(* CODESYS project P_ruwdkj.project
   Title: B_Ugol
   Version: 0.0.0.0

Project tree, tasks and I/O mapping:
  MyController : TM241CEC24T/U, Schneider Electric, order no. TM241CEC24T/U, version 4.0.5.9
    application Application
      task MAST (cyclic, interval 20 ms, priority 15, watchdog 100 ms x 1) calls POU_Hand, POU_Auto, POU_Out, POU_Alarm, POU_testing
      global variables GVL
      program POU_Hand [LD]
      program POU_Out [LD]
      program POU_Auto [LD]
      Symbols
      program POU_Alarm [LD]
      program POU_testing [LD]
    DI : Digital Inputs, Schneider Electric, version 4.0.5.9
        input  iwDI_IW0 : WORD  // IW0
        input  i_AvStop : BOOL  // IW0.I0
        input  i_TZ_K1 : BOOL  // IW0.I1
        input  i_TZ_KR2 : BOOL  // IW0.I2
        input  i_Tros_K1 : BOOL  // IW0.I3
        input  i_Tros_KR2 : BOOL  // IW0.I4
        input  i_Di_Rezerv1 : BOOL  // IW0.I5
        input  i_Di_Rezerv2 : BOOL  // IW0.I6
        input  i_Di_Rezerv3 : BOOL  // IW0.I7
        input  i_Di_Rezerv4 : BOOL  // IW0.I8
        input  i_Di_Rezerv5 : BOOL  // IW0.I9
        input  i_Di_Rezerv6 : BOOL  // IW0.I10
        input  i_Di_Rezerv7 : BOOL  // IW0.I11
        input  i_Di_Rezerv8 : BOOL  // IW0.I12
        input  i_Di_Rezerv9 : BOOL  // IW0.I13
        input  ibDI_IB1 : BYTE  // IB1
    DQ : Digital Outputs, Schneider Electric, version 4.0.5.9
        output q_PuskK1 : BOOL  // QW0.Q0
        output q_PuskEP80 : BOOL  // QW0.Q1
        output q_PuskKR2_for : BOOL  // QW0.Q2
        output q_PuskKR2_rev : BOOL  // QW0.Q3
        output q_Zvonok : BOOL  // QW0.Q4
        output q_Red1 : BOOL  // QW0.Q5
        output q_Yellow1 : BOOL  // QW0.Q6
        output q_Green1 : BOOL  // QW0.Q7
        output q_Red2 : BOOL  // QW0.Q8
        output q_Yellow2 : BOOL  // QW0.Q9
        output qbDQ_QB1 : BYTE  // QB1
        unmapped channels: QW0
    Counters : Counters, Schneider Electric, version 4.0.5.9
    Pulse_Generators : Pulse Generators, Schneider Electric, version 4.0.5.9
    Cartridge_1 : Cartridge, Schneider Electric, version 4.0.5.9
    IO_Bus : IO bus - TM3, Schneider Electric, version 4.0.5.9
      Module_1 : TM3DQ8T/G, Schneider Electric, order no. TM3DQ8T/G, version 1.0.1.3
          output q_Green2 : BOOL  // QB0.Q0
          output q_Dq_Rezerv1 : BOOL  // QB0.Q1
          output q_Dq_Rezerv2 : BOOL  // QB0.Q2
          output q_Dq_Rezerv3 : BOOL  // QB0.Q3
          output q_Dq_Rezerv4 : BOOL  // QB0.Q4
          output q_Dq_Rezerv5 : BOOL  // QB0.Q5
          output q_Dq_Rezerv6 : BOOL  // QB0.Q6
          output q_Dq_Rezerv7 : BOOL  // QB0.Q7
          unmapped channels: QB0
      Module_2 : TM3AI8/G, Schneider Electric, order no. TM3AI8/G, version 1.0.0.16
          settings: KPI Configuration.KPI Configuration[0] = 35; KPI Configuration.KPI Configuration[1] = 35; KPI Configuration.KPI Configuration[2] = 35; KPI Configuration.KPI Configuration[3] = 35; KPI Configuration.KPI Configuration[8] = 160; KPI Configuration.KPI Configuration[9] = 15; KPI Configuration.KPI Configuration[10] = 160; KPI Configuration.KPI Configuration[11] = 15; KPI Configuration.KPI Configuration[12] = 160; KPI Configuration.KPI Configuration[13] = 15; KPI Configuration.KPI Configuration[14] = 160; KPI Configuration.KPI Configuration[15] = 15; KPI Configuration.KPI Configuration[24] = 32; KPI Configuration.KPI Configuration[25] = 78; KPI Configuration.KPI Configuration[26] = 32; KPI Configuration.KPI Configuration[27] = 78; KPI Configuration.KPI Configuration[28] = 32; KPI Configuration.KPI Configuration[29] = 78; KPI Configuration.KPI Configuration[30] = 32; KPI Configuration.KPI Configuration[31] = 78
          input  i_Uroven111 : INT  // IW0
          input  i_Uroven112 : INT  // IW1
          input  i_Uroven3 : INT  // IW2
          input  i_Uroven4 : INT  // IW3
          input  iiModule_2_IW4 : INT  // IW4
          input  iiModule_2_IW5 : INT  // IW5
          input  iiModule_2_IW6 : INT  // IW6
          input  iiModule_2_IW7 : INT  // IW7
          input  ibModule_2_IBStatusIW0 : BYTE  // IBStatusIW0
          input  ibModule_2_IBStatusIW1 : BYTE  // IBStatusIW1
          input  ibModule_2_IBStatusIW2 : BYTE  // IBStatusIW2
          input  ibModule_2_IBStatusIW3 : BYTE  // IBStatusIW3
          input  ibModule_2_IBStatusIW4 : BYTE  // IBStatusIW4
          input  ibModule_2_IBStatusIW5 : BYTE  // IBStatusIW5
          input  ibModule_2_IBStatusIW6 : BYTE  // IBStatusIW6
          input  ibModule_2_IBStatusIW7 : BYTE  // IBStatusIW7
    COM_Bus : COM bus, Schneider Electric, version 4.0.5.9
    Ethernet_1 : Ethernet Network, Schneider Electric, version 4.0.5.9
    Serial_Line_1 : Serial line, Schneider Electric, version 4.0.5.9
      SoMachine_Network_Manager : SoMachine-Network Manager, Schneider Electric, version 4.0.0.2
    Serial_Line_2 : Serial line, Schneider Electric, version 4.0.5.9
      Modbus_Manager : Modbus Manager, Schneider Electric, version 4.0.0.2
    CAN_1 : CANopen bus, Schneider Electric, version 4.0.5.9
      CANopen_Performance : CANopen Performance, Schneider Electric, order no. 1806, version 3.0.1.24
          settings: ConfigVersion = 50659584
        Pitatel1 : Altivar 312, Schneider Electric, order no. 0, version 4.5.0.0
            settings: General Options.Optional Device = TRUE; NODEIDSAVED = 1; SDO Timeout = 1000000; Explicit Deactivate PDOs = FALSE; EXPERTSETTINGS = True; Heartbeat-Producer Time = 200; PDO 16#1405.COBID = 16#0301; PDO 16#1805.COBID = 16#0281; Heartbeat-Consuming1.Heartbeat-Time = 300 ms; Drivecom command reg..Subindex = 16#00; Drivecom command reg..Subindex = 16#00; Frequency Reference.Subindex = 16#03; Target velocity.Index = 16#6042; Target velocity.Subindex = 16#00; Target velocity.ObjectLength = 16; Drivecom status register.Subindex = 16#00; Drivecom status register.Subindex = 16#00; Output frequency.Index = 16#2002; Output frequency.Subindex = 16#03; Output frequency.ObjectLength = 16; Motor Current.Index = 16#2002; Motor Current.Subindex = 16#05; Motor Current.ObjectLength = 16; SDO List.Set Guardtime.Index = 16#100C; SDO List.Set Guardtime.Subindex = 16#00; SDO List.Set Guardtime.Value = 16#00000000; SDO List.Set Guardtime.Size = 16; SDO List.Set Guardtime.AbortIfError = FALSE; SDO List.Set Guardtime.JumpToLine = FALSE; SDO List.Set Guardtime.Line = 0; SDO List.Set Lifetime.Index = 16#100D; SDO List.Set Lifetime.Subindex = 16#00; SDO List.Set Lifetime.Value = 16#00000000; SDO List.Set Lifetime.Size = 8; SDO List.Set Lifetime.AbortIfError = FALSE; SDO List.Set Lifetime.JumpToLine = FALSE; SDO List.Set Lifetime.Line = 0; SDO List.Set Heartbeat Consumer.Index = 16#1016; SDO List.Set Heartbeat Consumer.Subindex = 16#01; SDO List.Set Heartbeat Consumer.Value = 16#007F012C;
              SDO List.Set Heartbeat Consumer.Size = 32; SDO List.Set Heartbeat Consumer.AbortIfError = FALSE; SDO List.Set Heartbeat Consumer.JumpToLine = FALSE; SDO List.Set Heartbeat Consumer.Line = 0; SDO List.Set Heartbeat Producer.Index = 16#1017; SDO List.Set Heartbeat Producer.Subindex = 16#00; SDO List.Set Heartbeat Producer.Value = 16#000000C8; SDO List.Set Heartbeat Producer.Size = 16; SDO List.Set Heartbeat Producer.AbortIfError = FALSE; SDO List.Set Heartbeat Producer.JumpToLine = FALSE; SDO List.Set Heartbeat Producer.Line = 0; SDO List.Disable PDO.Index = 16#1400; SDO List.Disable PDO.Subindex = 16#01; SDO List.Disable PDO.Value = 16#80000201; SDO List.Disable PDO.Size = 32; SDO List.Disable PDO.AbortIfError = FALSE; SDO List.Disable PDO.JumpToLine = FALSE; SDO List.Disable PDO.Line = 0; SDO List.Disable PDO.Index = 16#1405; SDO List.Disable PDO.Subindex = 16#01; SDO List.Disable PDO.Value = 16#80000301; SDO List.Disable PDO.Size = 32; SDO List.Disable PDO.AbortIfError = FALSE; SDO List.Disable PDO.JumpToLine = FALSE; SDO List.Disable PDO.Line = 0; SDO List.Set transmission type.Index = 16#1405; SDO List.Set transmission type.Subindex = 16#02; SDO List.Set transmission type.Value = 16#FF; SDO List.Set transmission type.Size = 8; SDO List.Set transmission type.AbortIfError = FALSE; SDO List.Set transmission type.JumpToLine = FALSE; SDO List.Set transmission type.Line = 0; SDO List.Clear pdo mapping.Index = 16#1605; SDO List.Clear pdo mapping.Subindex = 16#00; SDO List.Clear pdo mapping.Value = 16#0; SDO List.Clear pdo mapping.Size = 8; SDO List.Clear pdo mapping.AbortIfError = FALSE; SDO List.Clear pdo mapping.JumpToLine = FALSE; SDO List.Clear pdo mapping.Line = 0; SDO List.Set Mapping.Index = 16#1605;
              SDO List.Set Mapping.Subindex = 16#01; SDO List.Set Mapping.Value = 16#60400010; SDO List.Set Mapping.Size = 32; SDO List.Set Mapping.AbortIfError = FALSE; SDO List.Set Mapping.JumpToLine = FALSE; SDO List.Set Mapping.Line = 0; SDO List.Set Mapping.Index = 16#1605; SDO List.Set Mapping.Subindex = 16#02; SDO List.Set Mapping.Value = 16#20370310; SDO List.Set Mapping.Size = 32; SDO List.Set Mapping.AbortIfError = FALSE; SDO List.Set Mapping.JumpToLine = FALSE; SDO List.Set Mapping.Line = 0; SDO List.Set Mapping.Index = 16#1605; SDO List.Set Mapping.Subindex = 16#03; SDO List.Set Mapping.Value = 16#60420010; SDO List.Set Mapping.Size = 32; SDO List.Set Mapping.AbortIfError = FALSE; SDO List.Set Mapping.JumpToLine = FALSE; SDO List.Set Mapping.Line = 0; SDO List.Set number of pdos.Index = 16#1605; SDO List.Set number of pdos.Subindex = 16#00; SDO List.Set number of pdos.Value = 16#03; SDO List.Set number of pdos.Size = 8; SDO List.Set number of pdos.AbortIfError = FALSE; SDO List.Set number of pdos.JumpToLine = FALSE; SDO List.Set number of pdos.Line = 0; SDO List.Set and enable COB-ID.Index = 16#1405; SDO List.Set and enable COB-ID.Subindex = 16#01; SDO List.Set and enable COB-ID.Value = 16#00000301; SDO List.Set and enable COB-ID.Size = 32; SDO List.Set and enable COB-ID.AbortIfError = FALSE; SDO List.Set and enable COB-ID.JumpToLine = FALSE; SDO List.Set and enable COB-ID.Line = 0; SDO List.Disable PDO.Index = 16#1800; SDO List.Disable PDO.Subindex = 16#01; SDO List.Disable PDO.Value = 16#80000181; SDO List.Disable PDO.Size = 32; SDO List.Disable PDO.AbortIfError = FALSE; SDO List.Disable PDO.JumpToLine = FALSE;
              SDO List.Disable PDO.Line = 0; SDO List.Disable PDO.Index = 16#1805; SDO List.Disable PDO.Subindex = 16#01; SDO List.Disable PDO.Value = 16#80000281; SDO List.Disable PDO.Size = 32; SDO List.Disable PDO.AbortIfError = FALSE; SDO List.Disable PDO.JumpToLine = FALSE; SDO List.Disable PDO.Line = 0; SDO List.Set transmission type.Index = 16#1805; SDO List.Set transmission type.Subindex = 16#02; SDO List.Set transmission type.Value = 16#FF; SDO List.Set transmission type.Size = 8; SDO List.Set transmission type.AbortIfError = FALSE; SDO List.Set transmission type.JumpToLine = FALSE; SDO List.Set transmission type.Line = 0; SDO List.Set inhibit time.Index = 16#1805; SDO List.Set inhibit time.Subindex = 16#03; SDO List.Set inhibit time.Value = 16#001E; SDO List.Set inhibit time.Size = 16; SDO List.Set inhibit time.AbortIfError = FALSE; SDO List.Set inhibit time.JumpToLine = FALSE; SDO List.Set inhibit time.Line = 0; SDO List.Set event time.Index = 16#1805; SDO List.Set event time.Subindex = 16#05; SDO List.Set event time.Value = 16#0064; SDO List.Set event time.Size = 16; SDO List.Set event time.AbortIfError = FALSE; SDO List.Set event time.JumpToLine = FALSE; SDO List.Set event time.Line = 0; SDO List.Clear pdo mapping.Index = 16#1A05; SDO List.Clear pdo mapping.Subindex = 16#00; SDO List.Clear pdo mapping.Value = 16#0; SDO List.Clear pdo mapping.Size = 8; SDO List.Clear pdo mapping.AbortIfError = FALSE; SDO List.Clear pdo mapping.JumpToLine = FALSE; SDO List.Clear pdo mapping.Line = 0; SDO List.Set Mapping.Index = 16#1A05; SDO List.Set Mapping.Subindex = 16#01; SDO List.Set Mapping.Value = 16#60410010; SDO List.Set Mapping.Size = 32;
              SDO List.Set Mapping.AbortIfError = FALSE; SDO List.Set Mapping.JumpToLine = FALSE; SDO List.Set Mapping.Line = 0; SDO List.Set Mapping.Index = 16#1A05; SDO List.Set Mapping.Subindex = 16#02; SDO List.Set Mapping.Value = 16#20020310; SDO List.Set Mapping.Size = 32; SDO List.Set Mapping.AbortIfError = FALSE; SDO List.Set Mapping.JumpToLine = FALSE; SDO List.Set Mapping.Line = 0; SDO List.Set Mapping.Index = 16#1A05; SDO List.Set Mapping.Subindex = 16#03; SDO List.Set Mapping.Value = 16#20020510; SDO List.Set Mapping.Size = 32; SDO List.Set Mapping.AbortIfError = FALSE; SDO List.Set Mapping.JumpToLine = FALSE; SDO List.Set Mapping.Line = 0; SDO List.Set number of pdos.Index = 16#1A05; SDO List.Set number of pdos.Subindex = 16#00; SDO List.Set number of pdos.Value = 16#03; SDO List.Set number of pdos.Size = 8; SDO List.Set number of pdos.AbortIfError = FALSE; SDO List.Set number of pdos.JumpToLine = FALSE; SDO List.Set number of pdos.Line = 0; SDO List.Set and enable COB-ID.Index = 16#1805; SDO List.Set and enable COB-ID.Subindex = 16#01; SDO List.Set and enable COB-ID.Value = 16#00000281; SDO List.Set and enable COB-ID.Size = 32; SDO List.Set and enable COB-ID.AbortIfError = FALSE; SDO List.Set and enable COB-ID.JumpToLine = FALSE; SDO List.Set and enable COB-ID.Line = 0; ConfigVersion = 50659584
            output q_ATVPit1_Controlword : UINT  // Drivecom command reg.
            output qiAltivar_312_1_Frequency_Reference : INT  // Frequency Reference
            output q_ATVPit1_WriteVelocity : INT  // Target velocity
            input  i_ATVPit1_Status : UINT  // Drivecom status register
            input  i_ATVPit1_OutFrec : INT  // Output frequency
            input  i_ATVPit1_OutCur : UINT  // Motor Current
        Pitatel2 : Altivar 312, Schneider Electric, order no. 0, version 4.5.0.0
            settings: General Options.Optional Device = TRUE; NODEIDSAVED = 3; SDO Timeout = 1000000; Explicit Deactivate PDOs = FALSE; EXPERTSETTINGS = True; Emergency-General Parameters.Emergency COBID = 16#83; Heartbeat-Producer Time = 200; PDO 16#1400.COBID = 16#80000203; PDO 16#1405.COBID = 16#0303; PDO 16#1800.COBID = 16#80000183; PDO 16#1805.COBID = 16#0283; Heartbeat-Consuming1.Heartbeat-Time = 300 ms; Drivecom command reg..Subindex = 16#00; Drivecom command reg..Subindex = 16#00; Frequency Reference.Subindex = 16#03; Target velocity.Index = 16#6042; Target velocity.Subindex = 16#00; Target velocity.ObjectLength = 16; Drivecom status register.Subindex = 16#00; Drivecom status register.Subindex = 16#00; Output frequency.Index = 16#2002; Output frequency.Subindex = 16#03; Output frequency.ObjectLength = 16; Motor Current.Index = 16#2002; Motor Current.Subindex = 16#05; Motor Current.ObjectLength = 16; SDO List.Set Guardtime.Index = 16#100C; SDO List.Set Guardtime.Subindex = 16#00; SDO List.Set Guardtime.Value = 16#00000000; SDO List.Set Guardtime.Size = 16; SDO List.Set Guardtime.AbortIfError = FALSE; SDO List.Set Guardtime.JumpToLine = FALSE; SDO List.Set Guardtime.Line = 0; SDO List.Set Lifetime.Index = 16#100D; SDO List.Set Lifetime.Subindex = 16#00; SDO List.Set Lifetime.Value = 16#00000000; SDO List.Set Lifetime.Size = 8; SDO List.Set Lifetime.AbortIfError = FALSE; SDO List.Set Lifetime.JumpToLine = FALSE; SDO List.Set Lifetime.Line = 0;
              SDO List.Set Heartbeat Consumer.Index = 16#1016; SDO List.Set Heartbeat Consumer.Subindex = 16#01; SDO List.Set Heartbeat Consumer.Value = 16#007F012C; SDO List.Set Heartbeat Consumer.Size = 32; SDO List.Set Heartbeat Consumer.AbortIfError = FALSE; SDO List.Set Heartbeat Consumer.JumpToLine = FALSE; SDO List.Set Heartbeat Consumer.Line = 0; SDO List.Set Heartbeat Producer.Index = 16#1017; SDO List.Set Heartbeat Producer.Subindex = 16#00; SDO List.Set Heartbeat Producer.Value = 16#000000C8; SDO List.Set Heartbeat Producer.Size = 16; SDO List.Set Heartbeat Producer.AbortIfError = FALSE; SDO List.Set Heartbeat Producer.JumpToLine = FALSE; SDO List.Set Heartbeat Producer.Line = 0; SDO List.Disable PDO.Index = 16#1400; SDO List.Disable PDO.Subindex = 16#01; SDO List.Disable PDO.Value = 16#80000203; SDO List.Disable PDO.Size = 32; SDO List.Disable PDO.AbortIfError = FALSE; SDO List.Disable PDO.JumpToLine = FALSE; SDO List.Disable PDO.Line = 0; SDO List.Disable PDO.Index = 16#1405; SDO List.Disable PDO.Subindex = 16#01; SDO List.Disable PDO.Value = 16#80000303; SDO List.Disable PDO.Size = 32; SDO List.Disable PDO.AbortIfError = FALSE; SDO List.Disable PDO.JumpToLine = FALSE; SDO List.Disable PDO.Line = 0; SDO List.Set transmission type.Index = 16#1405; SDO List.Set transmission type.Subindex = 16#02; SDO List.Set transmission type.Value = 16#FF; SDO List.Set transmission type.Size = 8; SDO List.Set transmission type.AbortIfError = FALSE; SDO List.Set transmission type.JumpToLine = FALSE; SDO List.Set transmission type.Line = 0; SDO List.Clear pdo mapping.Index = 16#1605; SDO List.Clear pdo mapping.Subindex = 16#00; SDO List.Clear pdo mapping.Value = 16#0; SDO List.Clear pdo mapping.Size = 8; SDO List.Clear pdo mapping.AbortIfError = FALSE;
              SDO List.Clear pdo mapping.JumpToLine = FALSE; SDO List.Clear pdo mapping.Line = 0; SDO List.Set Mapping.Index = 16#1605; SDO List.Set Mapping.Subindex = 16#01; SDO List.Set Mapping.Value = 16#60400010; SDO List.Set Mapping.Size = 32; SDO List.Set Mapping.AbortIfError = FALSE; SDO List.Set Mapping.JumpToLine = FALSE; SDO List.Set Mapping.Line = 0; SDO List.Set Mapping.Index = 16#1605; SDO List.Set Mapping.Subindex = 16#02; SDO List.Set Mapping.Value = 16#20370310; SDO List.Set Mapping.Size = 32; SDO List.Set Mapping.AbortIfError = FALSE; SDO List.Set Mapping.JumpToLine = FALSE; SDO List.Set Mapping.Line = 0; SDO List.Set Mapping.Index = 16#1605; SDO List.Set Mapping.Subindex = 16#03; SDO List.Set Mapping.Value = 16#60420010; SDO List.Set Mapping.Size = 32; SDO List.Set Mapping.AbortIfError = FALSE; SDO List.Set Mapping.JumpToLine = FALSE; SDO List.Set Mapping.Line = 0; SDO List.Set number of pdos.Index = 16#1605; SDO List.Set number of pdos.Subindex = 16#00; SDO List.Set number of pdos.Value = 16#03; SDO List.Set number of pdos.Size = 8; SDO List.Set number of pdos.AbortIfError = FALSE; SDO List.Set number of pdos.JumpToLine = FALSE; SDO List.Set number of pdos.Line = 0; SDO List.Set and enable COB-ID.Index = 16#1405; SDO List.Set and enable COB-ID.Subindex = 16#01; SDO List.Set and enable COB-ID.Value = 16#00000303; SDO List.Set and enable COB-ID.Size = 32; SDO List.Set and enable COB-ID.AbortIfError = FALSE; SDO List.Set and enable COB-ID.JumpToLine = FALSE; SDO List.Set and enable COB-ID.Line = 0; SDO List.Disable PDO.Index = 16#1800; SDO List.Disable PDO.Subindex = 16#01; SDO List.Disable PDO.Value = 16#80000183;
              SDO List.Disable PDO.Size = 32; SDO List.Disable PDO.AbortIfError = FALSE; SDO List.Disable PDO.JumpToLine = FALSE; SDO List.Disable PDO.Line = 0; SDO List.Disable PDO.Index = 16#1805; SDO List.Disable PDO.Subindex = 16#01; SDO List.Disable PDO.Value = 16#80000283; SDO List.Disable PDO.Size = 32; SDO List.Disable PDO.AbortIfError = FALSE; SDO List.Disable PDO.JumpToLine = FALSE; SDO List.Disable PDO.Line = 0; SDO List.Set transmission type.Index = 16#1805; SDO List.Set transmission type.Subindex = 16#02; SDO List.Set transmission type.Value = 16#FF; SDO List.Set transmission type.Size = 8; SDO List.Set transmission type.AbortIfError = FALSE; SDO List.Set transmission type.JumpToLine = FALSE; SDO List.Set transmission type.Line = 0; SDO List.Set inhibit time.Index = 16#1805; SDO List.Set inhibit time.Subindex = 16#03; SDO List.Set inhibit time.Value = 16#001E; SDO List.Set inhibit time.Size = 16; SDO List.Set inhibit time.AbortIfError = FALSE; SDO List.Set inhibit time.JumpToLine = FALSE; SDO List.Set inhibit time.Line = 0; SDO List.Set event time.Index = 16#1805; SDO List.Set event time.Subindex = 16#05; SDO List.Set event time.Value = 16#0064; SDO List.Set event time.Size = 16; SDO List.Set event time.AbortIfError = FALSE; SDO List.Set event time.JumpToLine = FALSE; SDO List.Set event time.Line = 0; SDO List.Clear pdo mapping.Index = 16#1A05; SDO List.Clear pdo mapping.Subindex = 16#00; SDO List.Clear pdo mapping.Value = 16#0; SDO List.Clear pdo mapping.Size = 8; SDO List.Clear pdo mapping.AbortIfError = FALSE; SDO List.Clear pdo mapping.JumpToLine = FALSE; SDO List.Clear pdo mapping.Line = 0; SDO List.Set Mapping.Index = 16#1A05;
              SDO List.Set Mapping.Subindex = 16#01; SDO List.Set Mapping.Value = 16#60410010; SDO List.Set Mapping.Size = 32; SDO List.Set Mapping.AbortIfError = FALSE; SDO List.Set Mapping.JumpToLine = FALSE; SDO List.Set Mapping.Line = 0; SDO List.Set Mapping.Index = 16#1A05; SDO List.Set Mapping.Subindex = 16#02; SDO List.Set Mapping.Value = 16#20020310; SDO List.Set Mapping.Size = 32; SDO List.Set Mapping.AbortIfError = FALSE; SDO List.Set Mapping.JumpToLine = FALSE; SDO List.Set Mapping.Line = 0; SDO List.Set Mapping.Index = 16#1A05; SDO List.Set Mapping.Subindex = 16#03; SDO List.Set Mapping.Value = 16#20020510; SDO List.Set Mapping.Size = 32; SDO List.Set Mapping.AbortIfError = FALSE; SDO List.Set Mapping.JumpToLine = FALSE; SDO List.Set Mapping.Line = 0; SDO List.Set number of pdos.Index = 16#1A05; SDO List.Set number of pdos.Subindex = 16#00; SDO List.Set number of pdos.Value = 16#03; SDO List.Set number of pdos.Size = 8; SDO List.Set number of pdos.AbortIfError = FALSE; SDO List.Set number of pdos.JumpToLine = FALSE; SDO List.Set number of pdos.Line = 0; SDO List.Set and enable COB-ID.Index = 16#1805; SDO List.Set and enable COB-ID.Subindex = 16#01; SDO List.Set and enable COB-ID.Value = 16#00000283; SDO List.Set and enable COB-ID.Size = 32; SDO List.Set and enable COB-ID.AbortIfError = FALSE; SDO List.Set and enable COB-ID.JumpToLine = FALSE; SDO List.Set and enable COB-ID.Line = 0; ConfigVersion = 50659584
            output q_ATVPit2_Controlword : UINT  // Drivecom command reg.
            output qiAltivar_312_2_Frequency_Reference : INT  // Frequency Reference
            output q_ATVPit2_WriteVelocity : INT  // Target velocity
            input  i_ATVPit2_Status : UINT  // Drivecom status register
            input  i_ATVPit2_OutFrec : INT  // Output frequency
            input  i_ATVPit2_OutCur : UINT  // Motor Current
  HMIGTO3510 : HMIGTO3510, Schneider Electric, order no. HMIGTO3510, version 3.5.3.55
    HMI Application
    COM1
      SoMachine_Network_Manager1 : SoMachine-Network Manager, Schneider Electric, version 4.0.0.2
    COM2
      SoMachine_Network_Manager2 : SoMachine-Network Manager, Schneider Electric, version 4.0.0.2
    Ethernet
      SoMachine_Network_Manager3 : SoMachine-Network Manager, Schneider Electric, version 4.0.0.2
    USB
      SoMachine_Network_Manager4 : SoMachine-Network Manager, Schneider Electric, version 4.0.0.2
  6c0f7fb6-600b-4c93-9262-20cdc603757e
  Vijeo Designer Project Container
*)

// MyController/Application/GVL
VAR_GLOBAL
	// Маркер включения К-1 в ручном режиме
	Pusk_K1_RR: BOOL;
	// Маркер включения ЭП 80 в ручном режиме
	Pusk_EP80_RR: BOOL;
	// Маркер включения КР-2 прямо в ручном режиме
	Pusk_KR2for_RR: BOOL;
	// Маркер включения КР-2 реверс в ручном режиме
	Pusk_KR2rev_RR: BOOL;
	// Маркер включения ПЧ питателя 1.1.1 в ручном режиме
	Pusk_Pit1_RR: BOOL;
	// Маркер включения ПЧ питателя 1.1.2 в ручном режиме
	Pusk_Pit2_RR: BOOL;
	// Защита ПЧ питателя 1.1.1
	AvarATVPit1: BOOL;
	// Защита ПЧ питателя 1.1.2
	AvarATVPit2: BOOL;
	// Маркер включения звонка в ручном режиме
	Pusk_Zvonok_RR: BOOL;
	// Маркер включения первого звонка перед пусками в ручном режиме
	Zvonok1_RR: BOOL;
	// Маркер включения второго звонка перед пусками в ручном режиме
	Zvonok2_RR: BOOL;
	// Квитирование из панели
	KvitirHMI: BOOL;
	// Сводный маркер защит К-1
	Avar_K1: BOOL;
	// Маркер включения звонка при защитах
	Zvonok_Alarm: BOOL;
	// Фиксация Аварийного стопа
	AvarStop: BOOL;
	// Сводный маркер защит КР-2
	Avar_KR2: BOOL;
	// Сводный маркер защит питателя 1.1.1
	AvarPit1: BOOL;
	// Сводный маркер защит питателя 1.1.2
	AvarPit2: BOOL;
	// Маркер включения первого звонка перед пусками в авто режиме
	Zvonok1_AR: BOOL;
	// Маркер включения второго звонка перед пусками в авто режиме
	Zvonok2_AR: BOOL;
	// Маркер включения ЭП 80 в автоматическом режиме
	Pusk_EP80_AR: BOOL;
	// Маркер включения К-1 в автоматическом режиме
	Pusk_K1_AR: BOOL;
	// Маркер включения КР-2 прямо в автоматическом режиме
	Pusk_KR2for_AR: BOOL;
	// Маркер включения КР-2 реверс в автоматическом режиме
	Pusk_KR2rev_AR: BOOL;
	// Маркер включения ПЧ питателя 1.1.1 в автоматическом режиме
	Pusk_Pit1_AR: BOOL;
	// Маркер включения ПЧ питателя 1.1.2 в автоматическом режиме
	Pusk_Pit2_AR: BOOL;
	// Маркер максимального уровня в питателе 1.1.1
	Ur111_MAX: BOOL;
	// Маркер минимального уровня в питателе 1.1.1
	Ur111_MIN: BOOL;
	// Маркер среднего уровня в питателе 1.1.1
	Ur111_MIDL: BOOL;
	// Маркер минимального уровня в питателе 1.1.2
	Ur112_MIN: BOOL;
	// Маркер среднего уровня в питателе 1.1.2
	Ur112_MIDL: BOOL;
	// Маркер максимального уровня в питателе 1.1.2
	Ur112_MAX: BOOL;
	// Сводный маркер всех защит
	Avar_ALL: BOOL;
END_VAR

// MyController/Application/POU_Hand
PROGRAM POU_Hand
VAR
	// Маркер пуск из HMI К-1 в ручном режиме
	PuskHMI_K1_RR: BOOL;
	// Маркер пуск из HMI ЭП 80 в ручном режиме
	PuskHMI_EP80_RR: BOOL;
	// Маркер пуск из HMI КР-2 прямо в ручном режиме
	PuskHMI_KR2for_RR: BOOL;
	// Маркер пуск из HMI КР-2 реверс в ручном режиме
	PuskHMI_KR2rev_RR: BOOL;
	// Маркер пуск из HMI ПЧ питателя 1.1.1 в ручном режиме
	PuskHMI_Pit1_RR: BOOL;
	TP_ZV1: TP;
	TP_ZV2: TP;
	TP_ZV3: TP;
	// Маркер пуск из HMI ПЧ питателя 1.1.2 в ручном режиме
	PuskHMI_Pit2_RR: BOOL;
	// Маркер пуск из HMI звонка в ручном режиме
	PuskHMI_Zvonok_RR: BOOL;
	Pauza_RR: BOOL;
	// Маркер звонков перед пуском К-1 в РР
	ZvK1_RR: BOOL;
	// Маркер звонков перед пуском КР-2 прямо в РР
	ZvK2f_RR: BOOL;
	// Маркер звонков перед пуском КР-2 реверс в РР
	ZvK2r_RR: BOOL;
	// Маркер звонков перед пуском питателя 1 в РР
	ZvPit1_RR: BOOL;
	// Маркер звонков перед пуском питателя 2 в РР
	ZvPit2_RR: BOOL;
END_VAR
VAR // added by the converter: edge detectors and wires of the graphical bodies
    _rt1, _rt2, _rt3, _rt4, _rt5 : R_TRIG;
    _ft1, _ft2, _ft3, _ft4, _ft5, _ft6, _ft7 : F_TRIG;
END_VAR

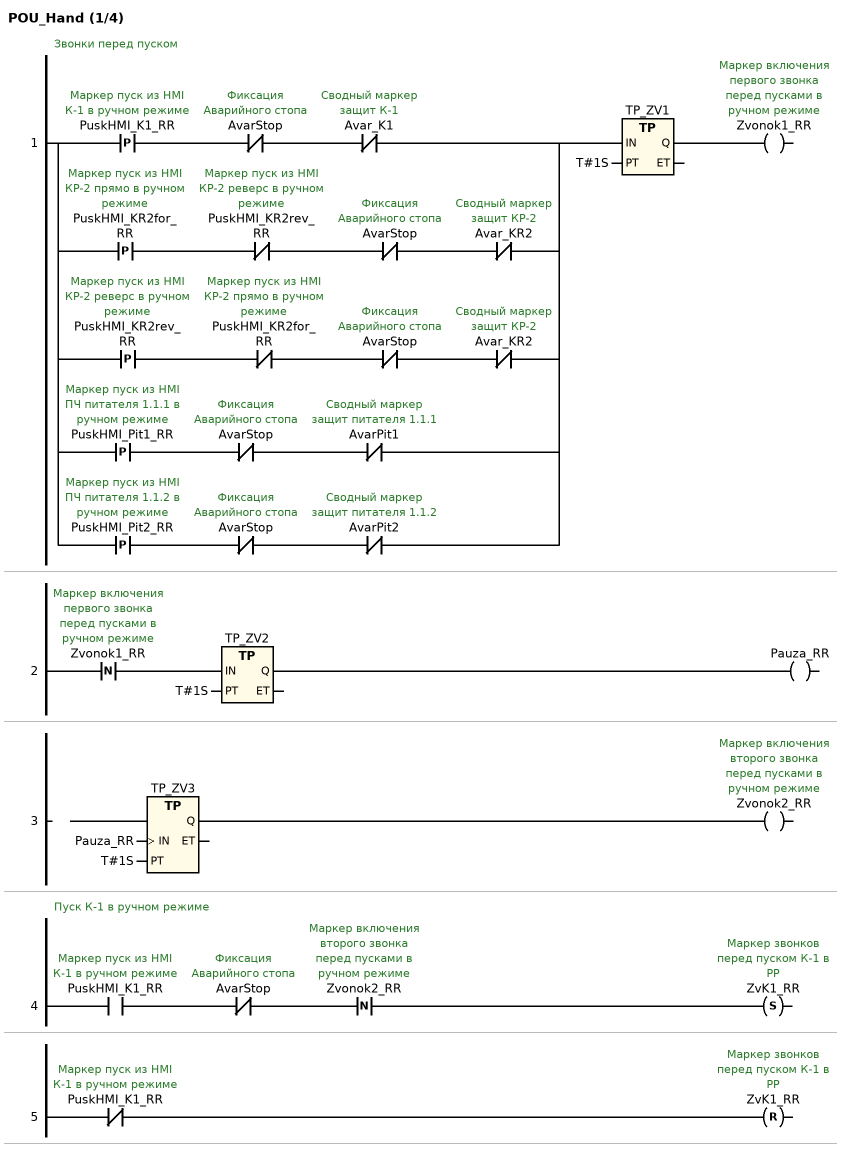
// NETWORK 1
// Звонки перед пуском
//   PuskHMI_K1_RR: Маркер пуск из HMI К-1 в ручном режиме
//   AvarStop: Фиксация Аварийного стопа
//   Avar_K1: Сводный маркер защит К-1
//   PuskHMI_KR2for_RR: Маркер пуск из HMI КР-2 прямо в ручном режиме
//   PuskHMI_KR2rev_RR: Маркер пуск из HMI КР-2 реверс в ручном режиме
//   Avar_KR2: Сводный маркер защит КР-2
//   PuskHMI_Pit1_RR: Маркер пуск из HMI ПЧ питателя 1.1.1 в ручном режиме
//   AvarPit1: Сводный маркер защит питателя 1.1.1
//   PuskHMI_Pit2_RR: Маркер пуск из HMI ПЧ питателя 1.1.2 в ручном режиме
//   AvarPit2: Сводный маркер защит питателя 1.1.2
//   Zvonok1_RR: Маркер включения первого звонка перед пусками в ручном режиме
_rt1(CLK := PuskHMI_K1_RR);
_rt2(CLK := PuskHMI_KR2for_RR);
_rt3(CLK := PuskHMI_KR2rev_RR);
_rt4(CLK := PuskHMI_Pit1_RR);
_rt5(CLK := PuskHMI_Pit2_RR);
TP_ZV1(IN := _rt1.Q AND NOT AvarStop AND NOT Avar_K1 OR _rt2.Q AND NOT PuskHMI_KR2rev_RR AND NOT AvarStop AND NOT Avar_KR2 OR _rt3.Q AND NOT PuskHMI_KR2for_RR AND NOT AvarStop AND NOT Avar_KR2 OR _rt4.Q AND NOT AvarStop AND NOT AvarPit1 OR _rt5.Q AND NOT AvarStop AND NOT AvarPit2, PT := T#1S); // TP
Zvonok1_RR := TP_ZV1.Q;

// NETWORK 2
//   Zvonok1_RR: Маркер включения первого звонка перед пусками в ручном режиме
_ft1(CLK := Zvonok1_RR);
TP_ZV2(IN := _ft1.Q, PT := T#1S); // TP
Pauza_RR := TP_ZV2.Q;

// NETWORK 3
//   Zvonok2_RR: Маркер включения второго звонка перед пусками в ручном режиме
_ft2(CLK := Pauza_RR);
TP_ZV3(IN := _ft2.Q, PT := T#1S); // TP
Zvonok2_RR := TP_ZV3.Q;

// NETWORK 4
// Пуск К-1 в ручном режиме
//   PuskHMI_K1_RR: Маркер пуск из HMI К-1 в ручном режиме
//   AvarStop: Фиксация Аварийного стопа
//   Zvonok2_RR: Маркер включения второго звонка перед пусками в ручном режиме
//   ZvK1_RR: Маркер звонков перед пуском К-1 в РР
_ft3(CLK := Zvonok2_RR);
ZvK1_RR S= PuskHMI_K1_RR AND NOT AvarStop AND _ft3.Q;

// NETWORK 5
//   PuskHMI_K1_RR: Маркер пуск из HMI К-1 в ручном режиме
//   ZvK1_RR: Маркер звонков перед пуском К-1 в РР
ZvK1_RR R= NOT PuskHMI_K1_RR;

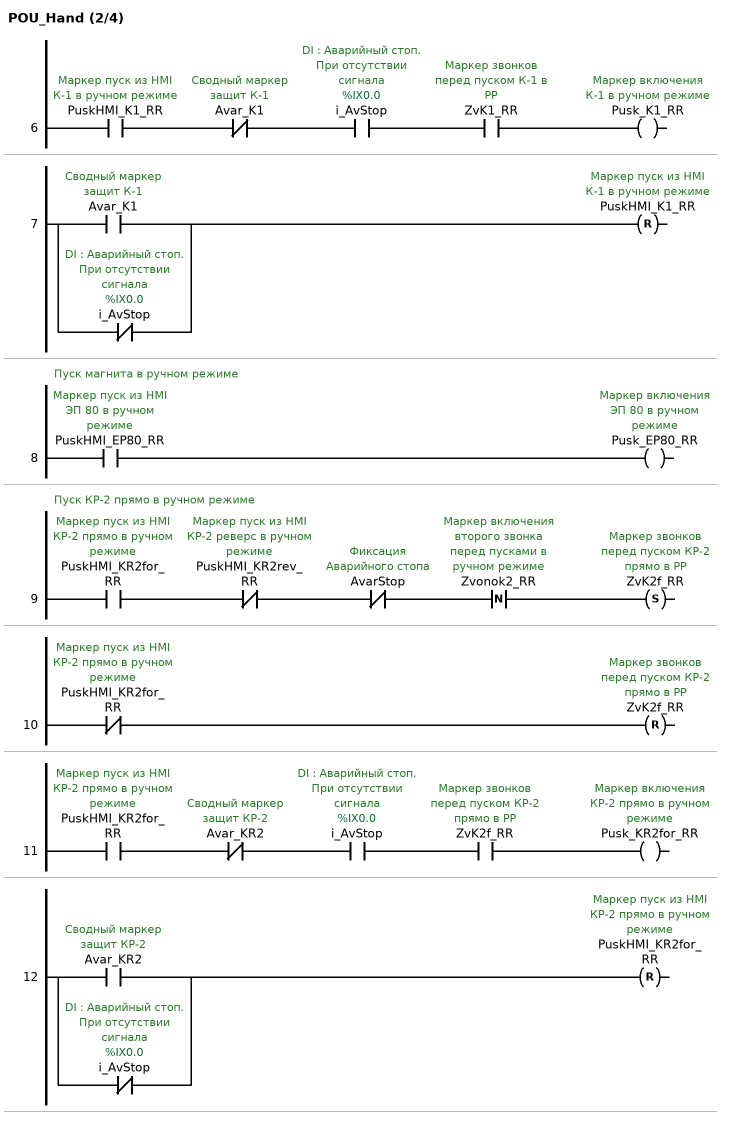
// NETWORK 6
//   PuskHMI_K1_RR: Маркер пуск из HMI К-1 в ручном режиме
//   Avar_K1: Сводный маркер защит К-1
//   i_AvStop: DI : Аварийный стоп. При отсутствии сигнала | AT %IX0.0
//   ZvK1_RR: Маркер звонков перед пуском К-1 в РР
//   Pusk_K1_RR: Маркер включения К-1 в ручном режиме
Pusk_K1_RR := PuskHMI_K1_RR AND NOT Avar_K1 AND i_AvStop AND ZvK1_RR;

// NETWORK 7
//   Avar_K1: Сводный маркер защит К-1
//   i_AvStop: DI : Аварийный стоп. При отсутствии сигнала | AT %IX0.0
//   PuskHMI_K1_RR: Маркер пуск из HMI К-1 в ручном режиме
PuskHMI_K1_RR R= Avar_K1 OR NOT i_AvStop;

// NETWORK 8
// Пуск магнита в ручном режиме
//   PuskHMI_EP80_RR: Маркер пуск из HMI ЭП 80 в ручном режиме
//   Pusk_EP80_RR: Маркер включения ЭП 80 в ручном режиме
Pusk_EP80_RR := PuskHMI_EP80_RR;

// NETWORK 9
// Пуск КР-2 прямо в ручном режиме
//   PuskHMI_KR2for_RR: Маркер пуск из HMI КР-2 прямо в ручном режиме
//   PuskHMI_KR2rev_RR: Маркер пуск из HMI КР-2 реверс в ручном режиме
//   AvarStop: Фиксация Аварийного стопа
//   Zvonok2_RR: Маркер включения второго звонка перед пусками в ручном режиме
//   ZvK2f_RR: Маркер звонков перед пуском КР-2 прямо в РР
_ft4(CLK := Zvonok2_RR);
ZvK2f_RR S= PuskHMI_KR2for_RR AND NOT PuskHMI_KR2rev_RR AND NOT AvarStop AND _ft4.Q;

// NETWORK 10
//   PuskHMI_KR2for_RR: Маркер пуск из HMI КР-2 прямо в ручном режиме
//   ZvK2f_RR: Маркер звонков перед пуском КР-2 прямо в РР
ZvK2f_RR R= NOT PuskHMI_KR2for_RR;

// NETWORK 11
//   PuskHMI_KR2for_RR: Маркер пуск из HMI КР-2 прямо в ручном режиме
//   Avar_KR2: Сводный маркер защит КР-2
//   i_AvStop: DI : Аварийный стоп. При отсутствии сигнала | AT %IX0.0
//   ZvK2f_RR: Маркер звонков перед пуском КР-2 прямо в РР
//   Pusk_KR2for_RR: Маркер включения КР-2 прямо в ручном режиме
Pusk_KR2for_RR := PuskHMI_KR2for_RR AND NOT Avar_KR2 AND i_AvStop AND ZvK2f_RR;

// NETWORK 12
//   Avar_KR2: Сводный маркер защит КР-2
//   i_AvStop: DI : Аварийный стоп. При отсутствии сигнала | AT %IX0.0
//   PuskHMI_KR2for_RR: Маркер пуск из HMI КР-2 прямо в ручном режиме
PuskHMI_KR2for_RR R= Avar_KR2 OR NOT i_AvStop;

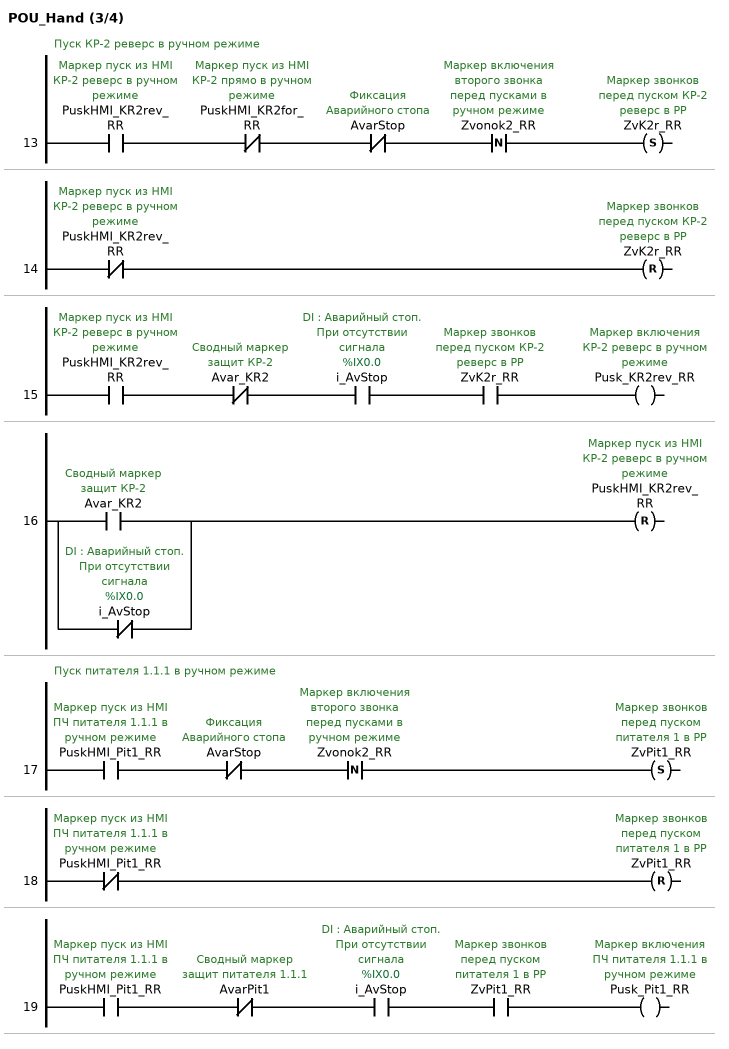
// NETWORK 13
// Пуск КР-2 реверс в ручном режиме
//   PuskHMI_KR2rev_RR: Маркер пуск из HMI КР-2 реверс в ручном режиме
//   PuskHMI_KR2for_RR: Маркер пуск из HMI КР-2 прямо в ручном режиме
//   AvarStop: Фиксация Аварийного стопа
//   Zvonok2_RR: Маркер включения второго звонка перед пусками в ручном режиме
//   ZvK2r_RR: Маркер звонков перед пуском КР-2 реверс в РР
_ft5(CLK := Zvonok2_RR);
ZvK2r_RR S= PuskHMI_KR2rev_RR AND NOT PuskHMI_KR2for_RR AND NOT AvarStop AND _ft5.Q;

// NETWORK 14
//   PuskHMI_KR2rev_RR: Маркер пуск из HMI КР-2 реверс в ручном режиме
//   ZvK2r_RR: Маркер звонков перед пуском КР-2 реверс в РР
ZvK2r_RR R= NOT PuskHMI_KR2rev_RR;

// NETWORK 15
//   PuskHMI_KR2rev_RR: Маркер пуск из HMI КР-2 реверс в ручном режиме
//   Avar_KR2: Сводный маркер защит КР-2
//   i_AvStop: DI : Аварийный стоп. При отсутствии сигнала | AT %IX0.0
//   ZvK2r_RR: Маркер звонков перед пуском КР-2 реверс в РР
//   Pusk_KR2rev_RR: Маркер включения КР-2 реверс в ручном режиме
Pusk_KR2rev_RR := PuskHMI_KR2rev_RR AND NOT Avar_KR2 AND i_AvStop AND ZvK2r_RR;

// NETWORK 16
//   Avar_KR2: Сводный маркер защит КР-2
//   i_AvStop: DI : Аварийный стоп. При отсутствии сигнала | AT %IX0.0
//   PuskHMI_KR2rev_RR: Маркер пуск из HMI КР-2 реверс в ручном режиме
PuskHMI_KR2rev_RR R= Avar_KR2 OR NOT i_AvStop;

// NETWORK 17
// Пуск питателя 1.1.1 в ручном режиме
//   PuskHMI_Pit1_RR: Маркер пуск из HMI ПЧ питателя 1.1.1 в ручном режиме
//   AvarStop: Фиксация Аварийного стопа
//   Zvonok2_RR: Маркер включения второго звонка перед пусками в ручном режиме
//   ZvPit1_RR: Маркер звонков перед пуском питателя 1 в РР
_ft6(CLK := Zvonok2_RR);
ZvPit1_RR S= PuskHMI_Pit1_RR AND NOT AvarStop AND _ft6.Q;

// NETWORK 18
//   PuskHMI_Pit1_RR: Маркер пуск из HMI ПЧ питателя 1.1.1 в ручном режиме
//   ZvPit1_RR: Маркер звонков перед пуском питателя 1 в РР
ZvPit1_RR R= NOT PuskHMI_Pit1_RR;

// NETWORK 19
//   PuskHMI_Pit1_RR: Маркер пуск из HMI ПЧ питателя 1.1.1 в ручном режиме
//   AvarPit1: Сводный маркер защит питателя 1.1.1
//   i_AvStop: DI : Аварийный стоп. При отсутствии сигнала | AT %IX0.0
//   ZvPit1_RR: Маркер звонков перед пуском питателя 1 в РР
//   Pusk_Pit1_RR: Маркер включения ПЧ питателя 1.1.1 в ручном режиме
Pusk_Pit1_RR := PuskHMI_Pit1_RR AND NOT AvarPit1 AND i_AvStop AND ZvPit1_RR;

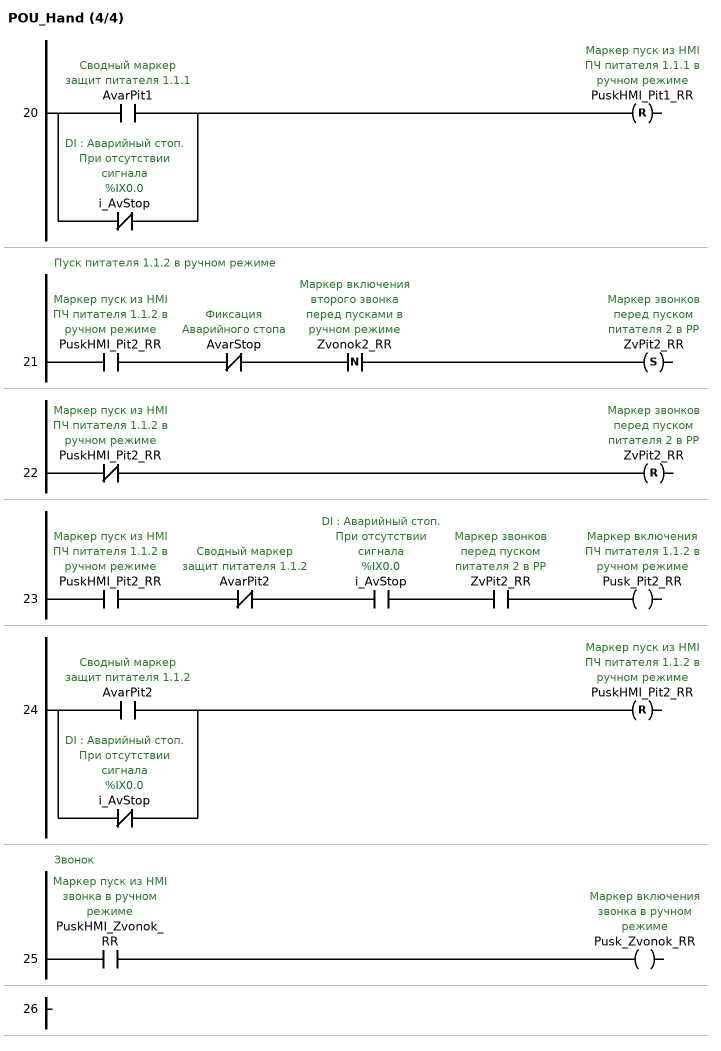
// NETWORK 20
//   AvarPit1: Сводный маркер защит питателя 1.1.1
//   i_AvStop: DI : Аварийный стоп. При отсутствии сигнала | AT %IX0.0
//   PuskHMI_Pit1_RR: Маркер пуск из HMI ПЧ питателя 1.1.1 в ручном режиме
PuskHMI_Pit1_RR R= AvarPit1 OR NOT i_AvStop;

// NETWORK 21
// Пуск питателя 1.1.2 в ручном режиме
//   PuskHMI_Pit2_RR: Маркер пуск из HMI ПЧ питателя 1.1.2 в ручном режиме
//   AvarStop: Фиксация Аварийного стопа
//   Zvonok2_RR: Маркер включения второго звонка перед пусками в ручном режиме
//   ZvPit2_RR: Маркер звонков перед пуском питателя 2 в РР
_ft7(CLK := Zvonok2_RR);
ZvPit2_RR S= PuskHMI_Pit2_RR AND NOT AvarStop AND _ft7.Q;

// NETWORK 22
//   PuskHMI_Pit2_RR: Маркер пуск из HMI ПЧ питателя 1.1.2 в ручном режиме
//   ZvPit2_RR: Маркер звонков перед пуском питателя 2 в РР
ZvPit2_RR R= NOT PuskHMI_Pit2_RR;

// NETWORK 23
//   PuskHMI_Pit2_RR: Маркер пуск из HMI ПЧ питателя 1.1.2 в ручном режиме
//   AvarPit2: Сводный маркер защит питателя 1.1.2
//   i_AvStop: DI : Аварийный стоп. При отсутствии сигнала | AT %IX0.0
//   ZvPit2_RR: Маркер звонков перед пуском питателя 2 в РР
//   Pusk_Pit2_RR: Маркер включения ПЧ питателя 1.1.2 в ручном режиме
Pusk_Pit2_RR := PuskHMI_Pit2_RR AND NOT AvarPit2 AND i_AvStop AND ZvPit2_RR;

// NETWORK 24
//   AvarPit2: Сводный маркер защит питателя 1.1.2
//   i_AvStop: DI : Аварийный стоп. При отсутствии сигнала | AT %IX0.0
//   PuskHMI_Pit2_RR: Маркер пуск из HMI ПЧ питателя 1.1.2 в ручном режиме
PuskHMI_Pit2_RR R= AvarPit2 OR NOT i_AvStop;

// NETWORK 25
// Звонок
//   PuskHMI_Zvonok_RR: Маркер пуск из HMI звонка в ручном режиме
//   Pusk_Zvonok_RR: Маркер включения звонка в ручном режиме
Pusk_Zvonok_RR := PuskHMI_Zvonok_RR;

// NETWORK 26

END_PROGRAM

// MyController/Application/POU_Auto
PROGRAM POU_Auto
VAR
	TP_ZV1a: TP;
	TP_ZV2a: TP;
	Pausa_AR: BOOL;
	TP_ZV3a: TP;
	// Пуск из HMI в автоматическом режиме
	PuskHMI_Auto: BOOL;
	// Маркер текущего уровня в % в питателе 1.1.1
	Ur111: INT;
	// Маркер выгрузки из питателя 1.1.1
	Vigruz111: BOOL;
	// Маркер текущего уровня в % в питателе 1.1.2
	Ur112: INT;
	// Маркер выгрузки из питателя 1.1.2
	Vigruz112: BOOL;
	// Маркер текущего уровня в % в бункере 3
	Ur3: INT;
	// Маркер максимального уровня в бункере 3
	Ur3_MAX: BOOL;
	// Маркер минимального уровня в бункере 3
	Ur3_MIN: BOOL;
	TON_K1_AR: TON;
	TON_Pit_AR: TON;
	RS_Vigruz111: RS;
	RS_Vigruz112: RS;
	RS_Auto: RS;
	// Маркер загрузки в бункер 3
	Zagruz3: BOOL;
	// Маркер текущего уровня в % в бункере 4
	Ur4: INT;
	// Маркер максимального уровня в бункере 4
	Ur4_MAX: BOOL;
	// Маркер минимального уровня в бункере 4
	Ur4_MIN: BOOL;
	// Маркер загрузки в бункер 4
	Zagruz4: BOOL;
	// Маркер автоматического пуска
	PuskAuto: BOOL;
	// Маркер отключения ЭП 80 в автоматическом режиме
	Stop_EP80_AR: BOOL;
	RS_Zagruz3: RS;
	RS_Zagruz4: RS;
	TON_Zagr3: TON;
	TON_Zagr4: TON;
	// Стоп автоматический из HMI
	StopAutoHMI: BOOL;
	// Стоп автоматический питателей
	StopAutoPit: BOOL;
	TOF_K1: TON;
	// Стоп автоматический К-1
	StopAutoK1: BOOL;
	TOF_KR2: TON;
	// Стоп автоматический КР-2
	StopAutoKR2: BOOL;
	TON_PAuto: TON;
	// Задержка выключения К-1 при автостопе
	OFF_K1: INT := 27;
	// Задержка выключения КР-2 при автостопе
	OFF_KR2: INT := 47;
END_VAR
VAR // added by the converter: edge detectors and wires of the graphical bodies
    _rt1 : R_TRIG;
    _ft1, _ft2, _ft3, _ft4 : F_TRIG;
    _w1 : BOOL;
END_VAR

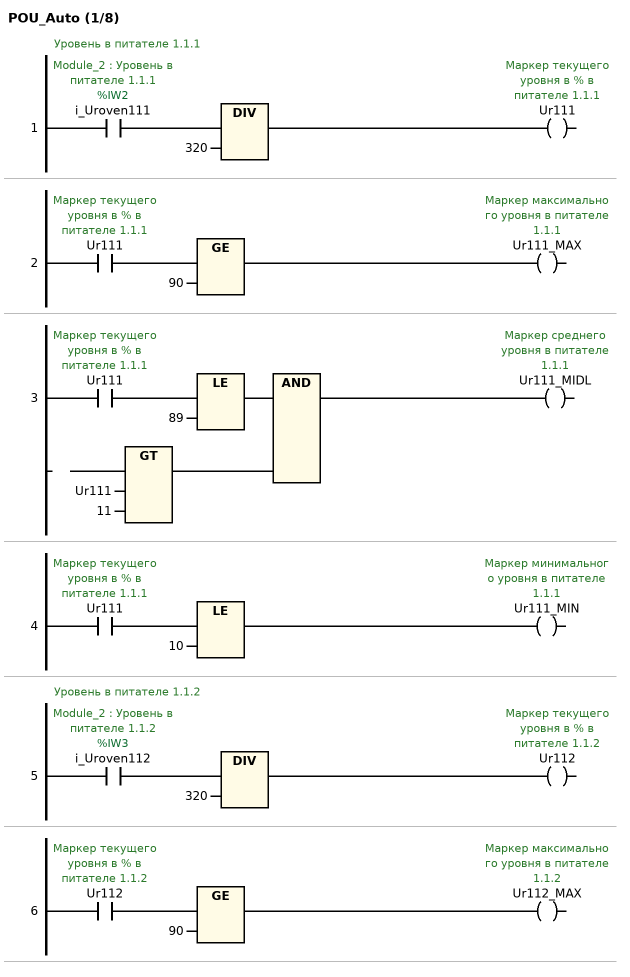
// NETWORK 1
// Уровень в питателе 1.1.1
//   i_Uroven111: Module_2 : Уровень в питателе 1.1.1 | AT %IW2
//   Ur111: Маркер текущего уровня в % в питателе 1.1.1
Ur111 := i_Uroven111 / 320;

// NETWORK 2
//   Ur111: Маркер текущего уровня в % в питателе 1.1.1
//   Ur111_MAX: Маркер максимального уровня в питателе 1.1.1
Ur111_MAX := Ur111 >= 90;

// NETWORK 3
//   Ur111: Маркер текущего уровня в % в питателе 1.1.1
//   Ur111_MIDL: Маркер среднего уровня в питателе 1.1.1
Ur111_MIDL := Ur111 <= 89 AND Ur111 > 11;

// NETWORK 4
//   Ur111: Маркер текущего уровня в % в питателе 1.1.1
//   Ur111_MIN: Маркер минимального уровня в питателе 1.1.1
Ur111_MIN := Ur111 <= 10;

// NETWORK 5
// Уровень в питателе 1.1.2
//   i_Uroven112: Module_2 : Уровень в питателе 1.1.2 | AT %IW3
//   Ur112: Маркер текущего уровня в % в питателе 1.1.2
Ur112 := i_Uroven112 / 320;

// NETWORK 6
//   Ur112: Маркер текущего уровня в % в питателе 1.1.2
//   Ur112_MAX: Маркер максимального уровня в питателе 1.1.2
Ur112_MAX := Ur112 >= 90;

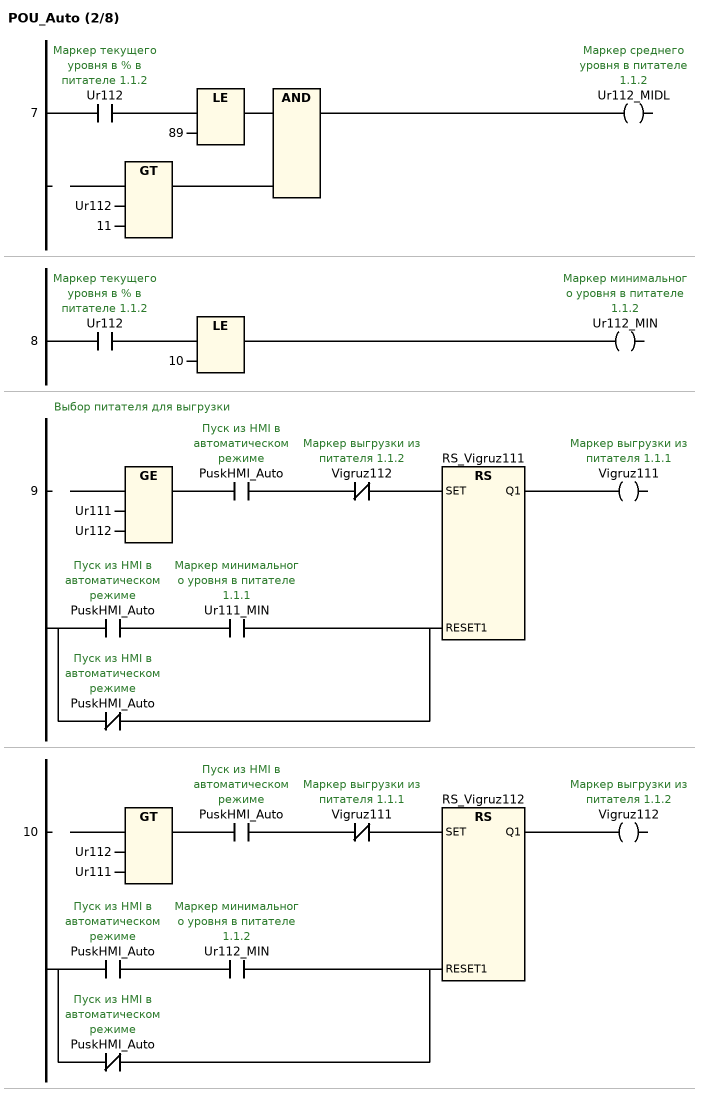
// NETWORK 7
//   Ur112: Маркер текущего уровня в % в питателе 1.1.2
//   Ur112_MIDL: Маркер среднего уровня в питателе 1.1.2
Ur112_MIDL := Ur112 <= 89 AND Ur112 > 11;

// NETWORK 8
//   Ur112: Маркер текущего уровня в % в питателе 1.1.2
//   Ur112_MIN: Маркер минимального уровня в питателе 1.1.2
Ur112_MIN := Ur112 <= 10;

// NETWORK 9
// Выбор питателя для выгрузки
//   Ur111: Маркер текущего уровня в % в питателе 1.1.1
//   Ur112: Маркер текущего уровня в % в питателе 1.1.2
//   PuskHMI_Auto: Пуск из HMI в автоматическом режиме
//   Vigruz112: Маркер выгрузки из питателя 1.1.2
//   Ur111_MIN: Маркер минимального уровня в питателе 1.1.1
//   Vigruz111: Маркер выгрузки из питателя 1.1.1
RS_Vigruz111(SET := Ur111 >= Ur112 AND PuskHMI_Auto AND NOT Vigruz112, RESET1 := PuskHMI_Auto AND Ur111_MIN OR NOT PuskHMI_Auto); // RS
Vigruz111 := RS_Vigruz111.Q1;

// NETWORK 10
//   Ur112: Маркер текущего уровня в % в питателе 1.1.2
//   Ur111: Маркер текущего уровня в % в питателе 1.1.1
//   PuskHMI_Auto: Пуск из HMI в автоматическом режиме
//   Vigruz111: Маркер выгрузки из питателя 1.1.1
//   Ur112_MIN: Маркер минимального уровня в питателе 1.1.2
//   Vigruz112: Маркер выгрузки из питателя 1.1.2
RS_Vigruz112(SET := Ur112 > Ur111 AND PuskHMI_Auto AND NOT Vigruz111, RESET1 := PuskHMI_Auto AND Ur112_MIN OR NOT PuskHMI_Auto); // RS
Vigruz112 := RS_Vigruz112.Q1;

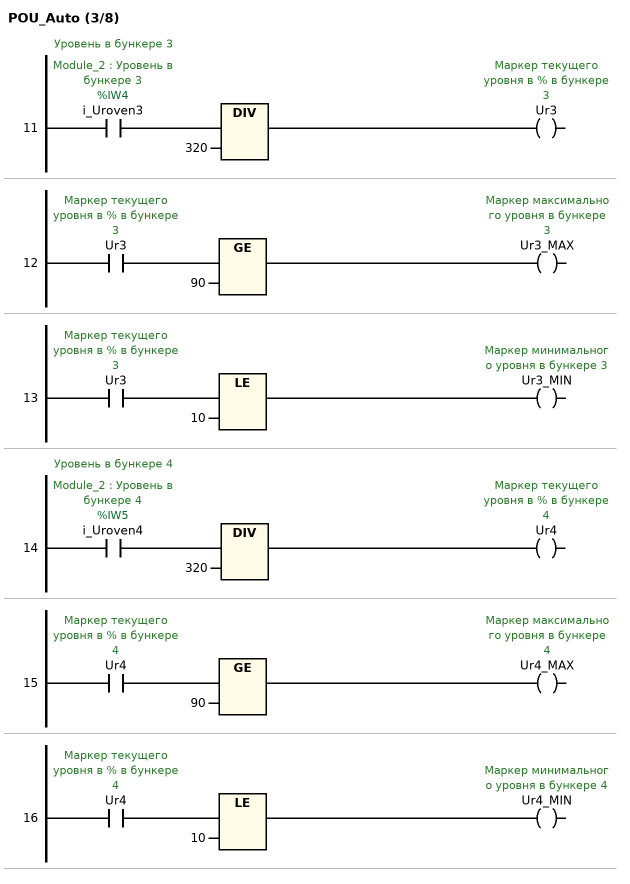
// NETWORK 11
// Уровень в бункере 3
//   i_Uroven3: Module_2 : Уровень в бункере 3 | AT %IW4
//   Ur3: Маркер текущего уровня в % в бункере 3
Ur3 := i_Uroven3 / 320;

// NETWORK 12
//   Ur3: Маркер текущего уровня в % в бункере 3
//   Ur3_MAX: Маркер максимального уровня в бункере 3
Ur3_MAX := Ur3 >= 90;

// NETWORK 13
//   Ur3: Маркер текущего уровня в % в бункере 3
//   Ur3_MIN: Маркер минимального уровня в бункере 3
Ur3_MIN := Ur3 <= 10;

// NETWORK 14
// Уровень в бункере 4
//   i_Uroven4: Module_2 : Уровень в бункере 4 | AT %IW5
//   Ur4: Маркер текущего уровня в % в бункере 4
Ur4 := i_Uroven4 / 320;

// NETWORK 15
//   Ur4: Маркер текущего уровня в % в бункере 4
//   Ur4_MAX: Маркер максимального уровня в бункере 4
Ur4_MAX := Ur4 >= 90;

// NETWORK 16
//   Ur4: Маркер текущего уровня в % в бункере 4
//   Ur4_MIN: Маркер минимального уровня в бункере 4
Ur4_MIN := Ur4 <= 10;

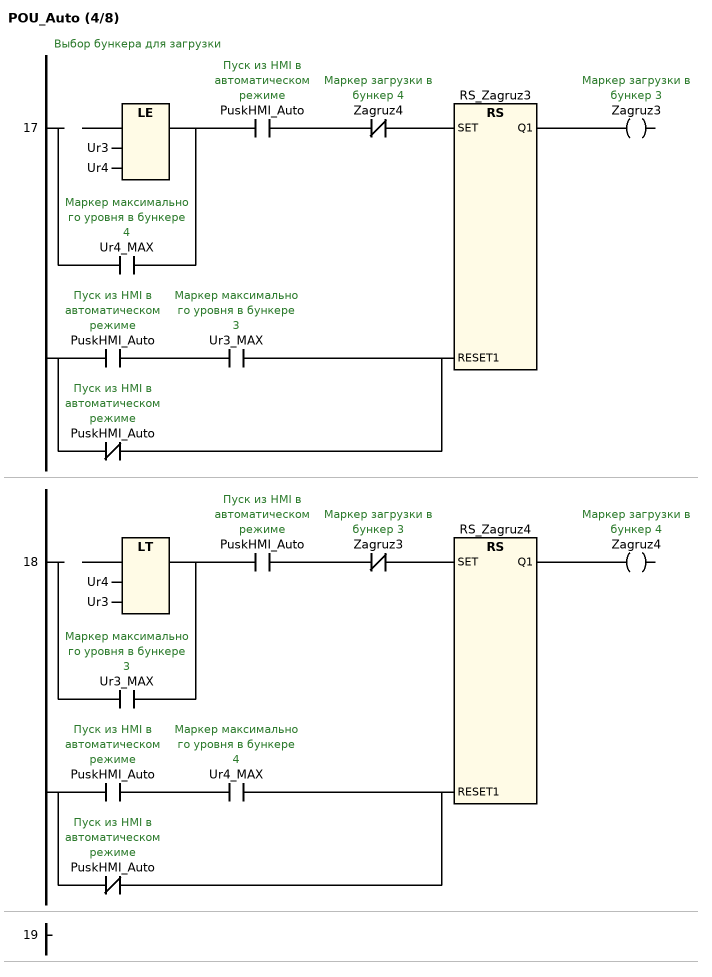
// NETWORK 17
// Выбор бункера для загрузки
//   Ur3: Маркер текущего уровня в % в бункере 3
//   Ur4: Маркер текущего уровня в % в бункере 4
//   Ur4_MAX: Маркер максимального уровня в бункере 4
//   PuskHMI_Auto: Пуск из HMI в автоматическом режиме
//   Zagruz4: Маркер загрузки в бункер 4
//   Ur3_MAX: Маркер максимального уровня в бункере 3
//   Zagruz3: Маркер загрузки в бункер 3
RS_Zagruz3(SET := (Ur3 <= Ur4 OR Ur4_MAX) AND PuskHMI_Auto AND NOT Zagruz4, RESET1 := PuskHMI_Auto AND Ur3_MAX OR NOT PuskHMI_Auto); // RS
Zagruz3 := RS_Zagruz3.Q1;

// NETWORK 18
//   Ur4: Маркер текущего уровня в % в бункере 4
//   Ur3: Маркер текущего уровня в % в бункере 3
//   Ur3_MAX: Маркер максимального уровня в бункере 3
//   PuskHMI_Auto: Пуск из HMI в автоматическом режиме
//   Zagruz3: Маркер загрузки в бункер 3
//   Ur4_MAX: Маркер максимального уровня в бункере 4
//   Zagruz4: Маркер загрузки в бункер 4
RS_Zagruz4(SET := (Ur4 < Ur3 OR Ur3_MAX) AND PuskHMI_Auto AND NOT Zagruz3, RESET1 := PuskHMI_Auto AND Ur4_MAX OR NOT PuskHMI_Auto); // RS
Zagruz4 := RS_Zagruz4.Q1;

// NETWORK 19

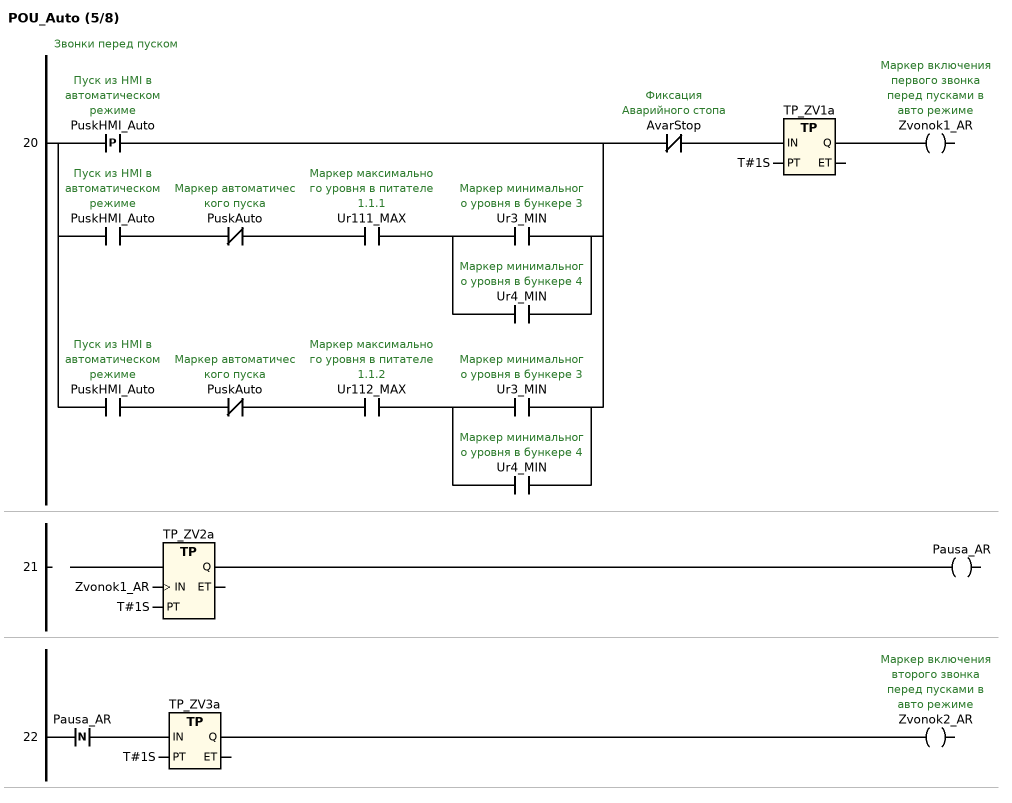
// NETWORK 20
// Звонки перед пуском
//   PuskHMI_Auto: Пуск из HMI в автоматическом режиме
//   PuskAuto: Маркер автоматического пуска
//   Ur111_MAX: Маркер максимального уровня в питателе 1.1.1
//   Ur3_MIN: Маркер минимального уровня в бункере 3
//   Ur4_MIN: Маркер минимального уровня в бункере 4
//   Ur112_MAX: Маркер максимального уровня в питателе 1.1.2
//   AvarStop: Фиксация Аварийного стопа
//   Zvonok1_AR: Маркер включения первого звонка перед пусками в авто режиме
_rt1(CLK := PuskHMI_Auto);
TP_ZV1a(IN := (_rt1.Q OR PuskHMI_Auto AND NOT PuskAuto AND Ur111_MAX AND (Ur3_MIN OR Ur4_MIN) OR PuskHMI_Auto AND NOT PuskAuto AND Ur112_MAX AND (Ur3_MIN OR Ur4_MIN)) AND NOT AvarStop, PT := T#1S); // TP
Zvonok1_AR := TP_ZV1a.Q;

// NETWORK 21
//   Zvonok1_AR: Маркер включения первого звонка перед пусками в авто режиме
_ft1(CLK := Zvonok1_AR);
TP_ZV2a(IN := _ft1.Q, PT := T#1S); // TP
Pausa_AR := TP_ZV2a.Q;

// NETWORK 22
//   Zvonok2_AR: Маркер включения второго звонка перед пусками в авто режиме
_ft2(CLK := Pausa_AR);
TP_ZV3a(IN := _ft2.Q, PT := T#1S); // TP
Zvonok2_AR := TP_ZV3a.Q;

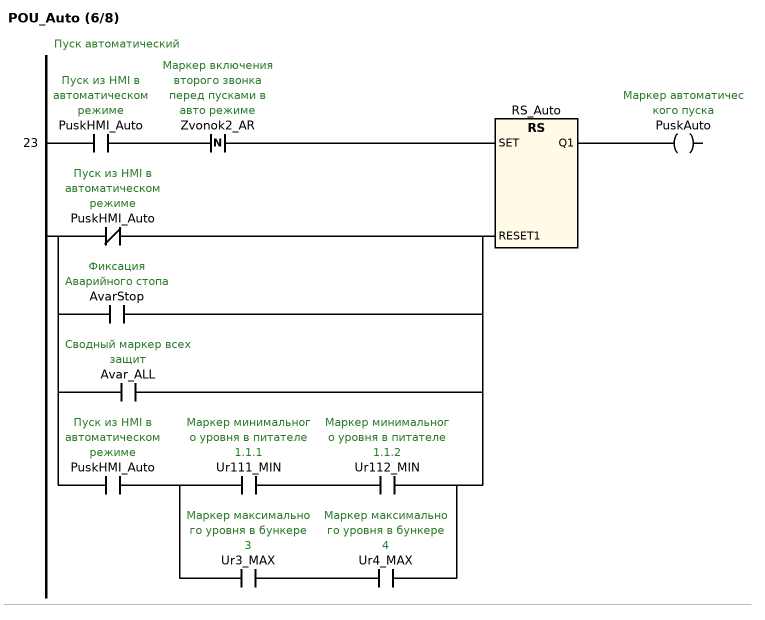
// NETWORK 23
// Пуск автоматический
//   PuskHMI_Auto: Пуск из HMI в автоматическом режиме
//   Zvonok2_AR: Маркер включения второго звонка перед пусками в авто режиме
//   AvarStop: Фиксация Аварийного стопа
//   Avar_ALL: Сводный маркер всех защит
//   Ur111_MIN: Маркер минимального уровня в питателе 1.1.1
//   Ur112_MIN: Маркер минимального уровня в питателе 1.1.2
//   Ur3_MAX: Маркер максимального уровня в бункере 3
//   Ur4_MAX: Маркер максимального уровня в бункере 4
//   PuskAuto: Маркер автоматического пуска
_ft3(CLK := Zvonok2_AR);
RS_Auto(SET := PuskHMI_Auto AND _ft3.Q, RESET1 := NOT PuskHMI_Auto OR AvarStop OR Avar_ALL OR PuskHMI_Auto AND (Ur111_MIN AND Ur112_MIN OR Ur3_MAX AND Ur4_MAX)); // RS
PuskAuto := RS_Auto.Q1;

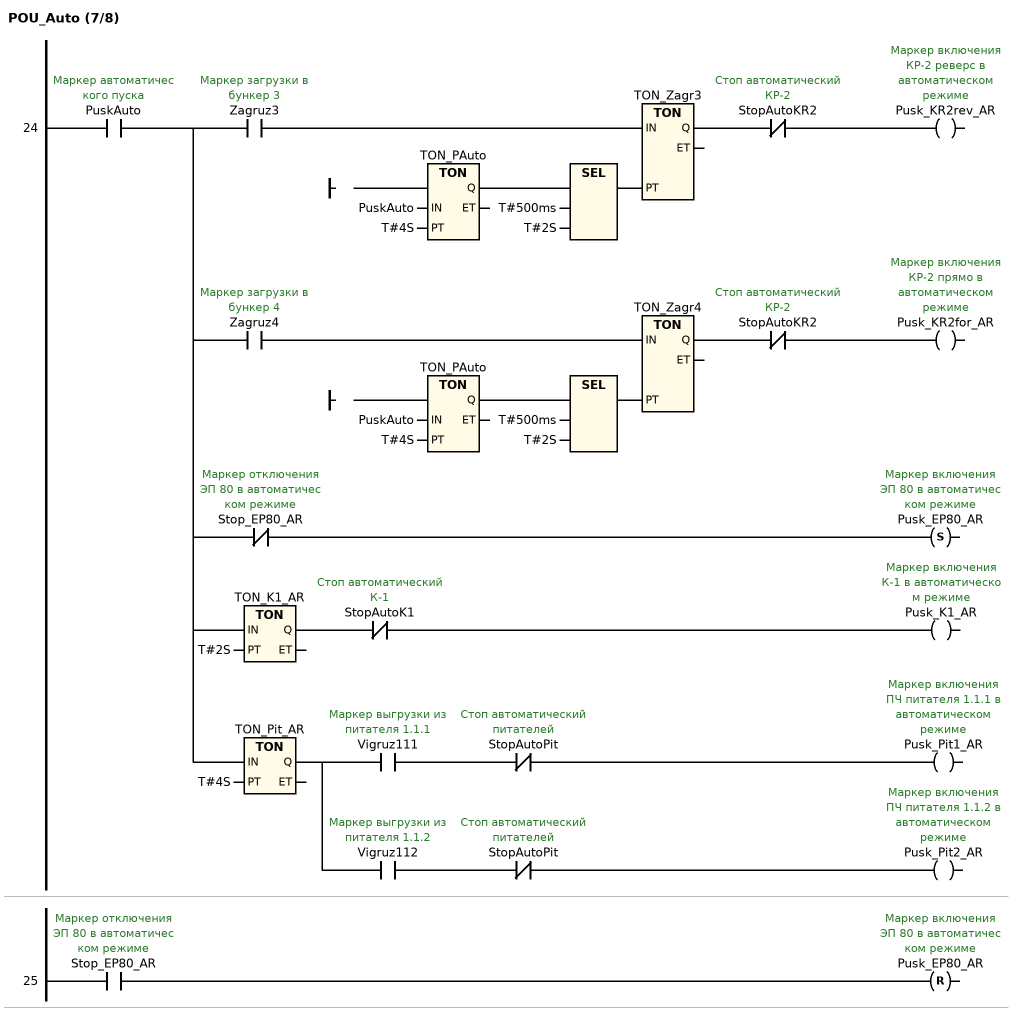
// NETWORK 24
//   PuskAuto: Маркер автоматического пуска
//   Zagruz3: Маркер загрузки в бункер 3
//   StopAutoKR2: Стоп автоматический КР-2
//   Pusk_KR2rev_AR: Маркер включения КР-2 реверс в автоматическом режиме
//   Zagruz4: Маркер загрузки в бункер 4
//   Pusk_KR2for_AR: Маркер включения КР-2 прямо в автоматическом режиме
//   Stop_EP80_AR: Маркер отключения ЭП 80 в автоматическом режиме
//   Pusk_EP80_AR: Маркер включения ЭП 80 в автоматическом режиме
//   StopAutoK1: Стоп автоматический К-1
//   Pusk_K1_AR: Маркер включения К-1 в автоматическом режиме
//   Vigruz111: Маркер выгрузки из питателя 1.1.1
//   StopAutoPit: Стоп автоматический питателей
//   Pusk_Pit1_AR: Маркер включения ПЧ питателя 1.1.1 в автоматическом режиме
//   Vigruz112: Маркер выгрузки из питателя 1.1.2
//   Pusk_Pit2_AR: Маркер включения ПЧ питателя 1.1.2 в автоматическом режиме
TON_PAuto(IN := PuskAuto, PT := T#4S); // TON
TON_Zagr3(IN := PuskAuto AND Zagruz3, PT := SEL(TON_PAuto.Q, T#500ms, T#2S)); // TON
Pusk_KR2rev_AR := TON_Zagr3.Q AND NOT StopAutoKR2;
TON_PAuto(IN := PuskAuto, PT := T#4S); // TON
TON_Zagr4(IN := PuskAuto AND Zagruz4, PT := SEL(TON_PAuto.Q, T#500ms, T#2S)); // TON
Pusk_KR2for_AR := TON_Zagr4.Q AND NOT StopAutoKR2;
Pusk_EP80_AR S= PuskAuto AND NOT Stop_EP80_AR;
TON_K1_AR(IN := PuskAuto, PT := T#2S); // TON
Pusk_K1_AR := TON_K1_AR.Q AND NOT StopAutoK1;
TON_Pit_AR(IN := PuskAuto, PT := T#4S); // TON
Pusk_Pit1_AR := TON_Pit_AR.Q AND Vigruz111 AND NOT StopAutoPit;
Pusk_Pit2_AR := TON_Pit_AR.Q AND Vigruz112 AND NOT StopAutoPit;

// NETWORK 25
//   Stop_EP80_AR: Маркер отключения ЭП 80 в автоматическом режиме
//   Pusk_EP80_AR: Маркер включения ЭП 80 в автоматическом режиме
Pusk_EP80_AR R= Stop_EP80_AR;

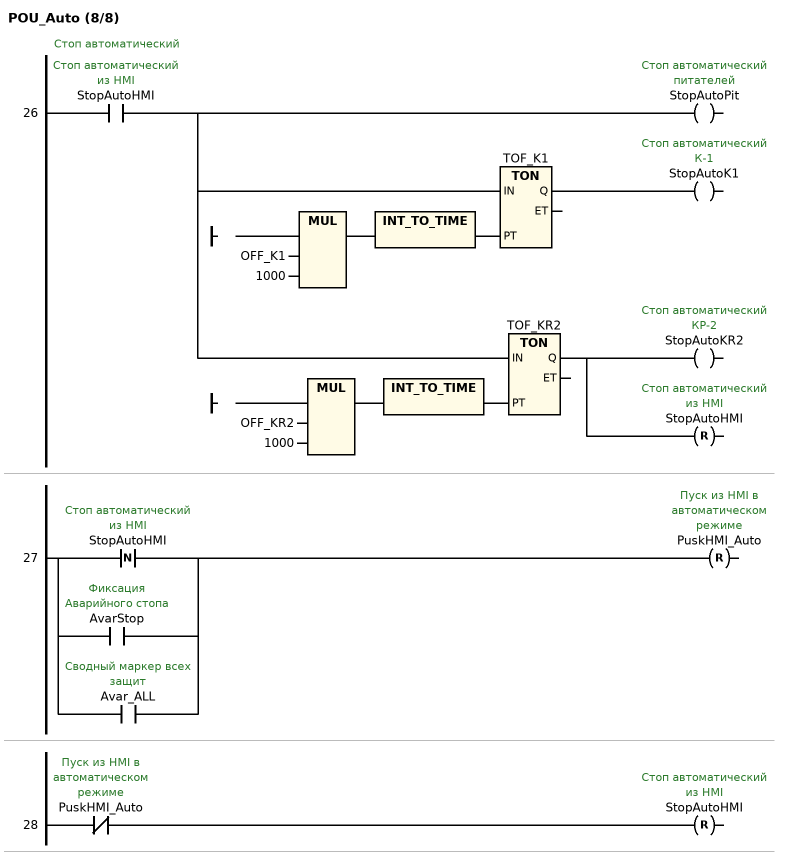
// NETWORK 26
// Стоп автоматический
//   StopAutoHMI: Стоп автоматический из HMI
//   StopAutoPit: Стоп автоматический питателей
//   OFF_K1: Задержка выключения К-1 при автостопе
//   StopAutoK1: Стоп автоматический К-1
//   OFF_KR2: Задержка выключения КР-2 при автостопе
//   StopAutoKR2: Стоп автоматический КР-2
_w1 := StopAutoHMI;
StopAutoPit := _w1;
TOF_K1(IN := _w1, PT := INT_TO_TIME(OFF_K1 * 1000)); // TON
StopAutoK1 := TOF_K1.Q;
TOF_KR2(IN := _w1, PT := INT_TO_TIME(OFF_KR2 * 1000)); // TON
StopAutoKR2 := TOF_KR2.Q;
StopAutoHMI R= TOF_KR2.Q;

// NETWORK 27
//   StopAutoHMI: Стоп автоматический из HMI
//   AvarStop: Фиксация Аварийного стопа
//   Avar_ALL: Сводный маркер всех защит
//   PuskHMI_Auto: Пуск из HMI в автоматическом режиме
_ft4(CLK := StopAutoHMI);
PuskHMI_Auto R= _ft4.Q OR AvarStop OR Avar_ALL;

// NETWORK 28
//   PuskHMI_Auto: Пуск из HMI в автоматическом режиме
//   StopAutoHMI: Стоп автоматический из HMI
StopAutoHMI R= NOT PuskHMI_Auto;

END_PROGRAM

// MyController/Application/POU_Out
PROGRAM POU_Out
VAR
	FB_ATV_Pit1: Altivar31_Control;
	FB_ATV_Pit2: Altivar31_Control;
	TON_ATV: TON;
	// Выходная частота питателя 1.1.1
	ATVPit1_OutFrec: INT;
	// Выходной ток питателя 1.1.1
	ATVPit1_OutCur: INT;
	// Задание из HMI частоты питателя 1.1.1
	ATVPit1_WriteFrecHMI: INT := 50;
	// Выходная частота питателя 1.1.2
	ATVPit2_OutFrec: INT;
	// Выходной ток питателя 1.1.2
	ATVPit2_OutCur: INT;
	// Задание из HMI частоты питателя 1.1.2
	ATVPit2_WriteFrecHMI: INT := 50;
	// Маркер пуск из HMI красный 1 в ручном режиме
	PuskHMI_Red1_RR: BOOL;
	// Маркер пуск из HMI желтый 1 в ручном режиме
	PuskHMI_Yellow1_RR: BOOL;
	// Маркер пуск из HMI зеленый 1 в ручном режиме
	PuskHMI_Green1_RR: BOOL;
	// Маркер пуск из HMI красный 2 в ручном режиме
	PuskHMI_Red2_RR: BOOL;
	// Маркер пуск из HMI желтый 2 в ручном режиме
	PuskHMI_Yellow2_RR: BOOL;
	// Маркер пуск из HMI зеленый 2 в ручном режиме
	PuskHMI_Green2_RR: BOOL;
END_VAR

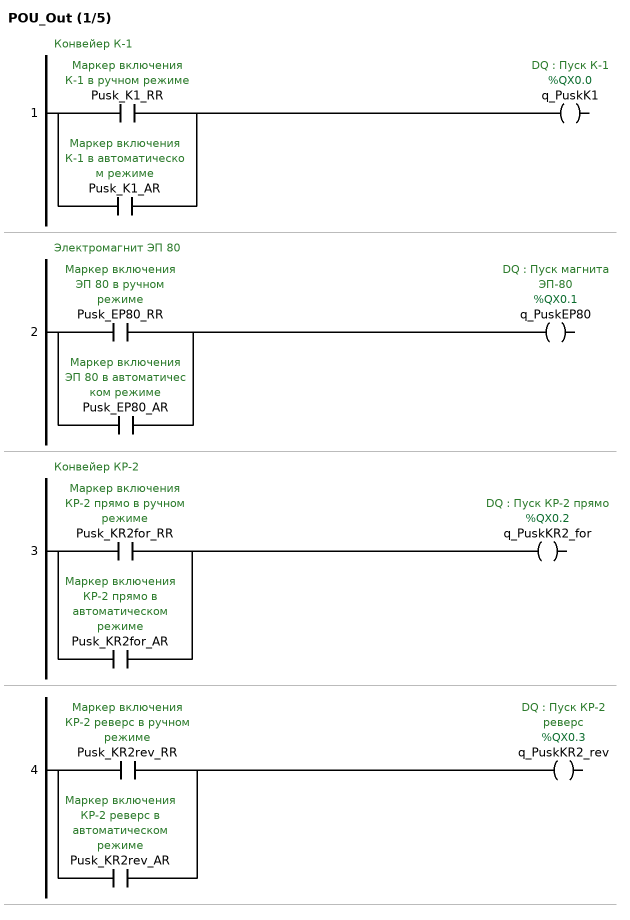
// NETWORK 1
// Конвейер К-1
//   Pusk_K1_RR: Маркер включения К-1 в ручном режиме
//   Pusk_K1_AR: Маркер включения К-1 в автоматическом режиме
//   q_PuskK1: DQ : Пуск К-1 | AT %QX0.0
q_PuskK1 := Pusk_K1_RR OR Pusk_K1_AR;

// NETWORK 2
// Электромагнит ЭП 80
//   Pusk_EP80_RR: Маркер включения ЭП 80 в ручном режиме
//   Pusk_EP80_AR: Маркер включения ЭП 80 в автоматическом режиме
//   q_PuskEP80: DQ : Пуск магнита ЭП-80 | AT %QX0.1
q_PuskEP80 := Pusk_EP80_RR OR Pusk_EP80_AR;

// NETWORK 3
// Конвейер КР-2
//   Pusk_KR2for_RR: Маркер включения КР-2 прямо в ручном режиме
//   Pusk_KR2for_AR: Маркер включения КР-2 прямо в автоматическом режиме
//   q_PuskKR2_for: DQ : Пуск КР-2 прямо | AT %QX0.2
q_PuskKR2_for := Pusk_KR2for_RR OR Pusk_KR2for_AR;

// NETWORK 4
//   Pusk_KR2rev_RR: Маркер включения КР-2 реверс в ручном режиме
//   Pusk_KR2rev_AR: Маркер включения КР-2 реверс в автоматическом режиме
//   q_PuskKR2_rev: DQ : Пуск КР-2 реверс | AT %QX0.3
q_PuskKR2_rev := Pusk_KR2rev_RR OR Pusk_KR2rev_AR;

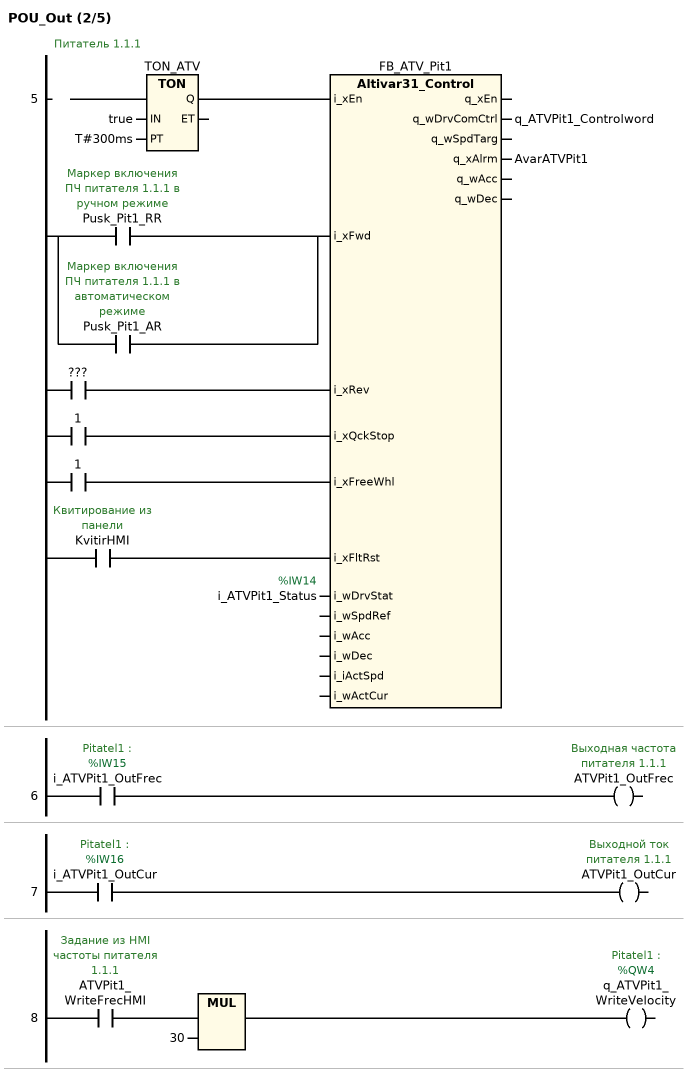
// NETWORK 5
// Питатель 1.1.1
//   Pusk_Pit1_RR: Маркер включения ПЧ питателя 1.1.1 в ручном режиме
//   Pusk_Pit1_AR: Маркер включения ПЧ питателя 1.1.1 в автоматическом режиме
//   KvitirHMI: Квитирование из панели
//   i_ATVPit1_Status: Pitatel1 : | AT %IW14
//   q_ATVPit1_Controlword: Pitatel1 : | AT %QW2
//   AvarATVPit1: Защита ПЧ питателя 1.1.1
TON_ATV(IN := true, PT := T#300ms); // TON
FB_ATV_Pit1(
    i_xEn := TON_ATV.Q,
    i_xFwd := Pusk_Pit1_RR OR Pusk_Pit1_AR,
    i_xQckStop := 1,
    i_xFreeWhl := 1,
    i_xFltRst := KvitirHMI,
    i_wDrvStat := i_ATVPit1_Status,
    q_wDrvComCtrl => q_ATVPit1_Controlword,
    q_xAlrm => AvarATVPit1); // Altivar31_Control

// NETWORK 6
//   i_ATVPit1_OutFrec: Pitatel1 : | AT %IW15
//   ATVPit1_OutFrec: Выходная частота питателя 1.1.1
ATVPit1_OutFrec := i_ATVPit1_OutFrec;

// NETWORK 7
//   i_ATVPit1_OutCur: Pitatel1 : | AT %IW16
//   ATVPit1_OutCur: Выходной ток питателя 1.1.1
ATVPit1_OutCur := i_ATVPit1_OutCur;

// NETWORK 8
//   ATVPit1_WriteFrecHMI: Задание из HMI частоты питателя 1.1.1
//   q_ATVPit1_WriteVelocity: Pitatel1 : | AT %QW4
q_ATVPit1_WriteVelocity := ATVPit1_WriteFrecHMI * 30;

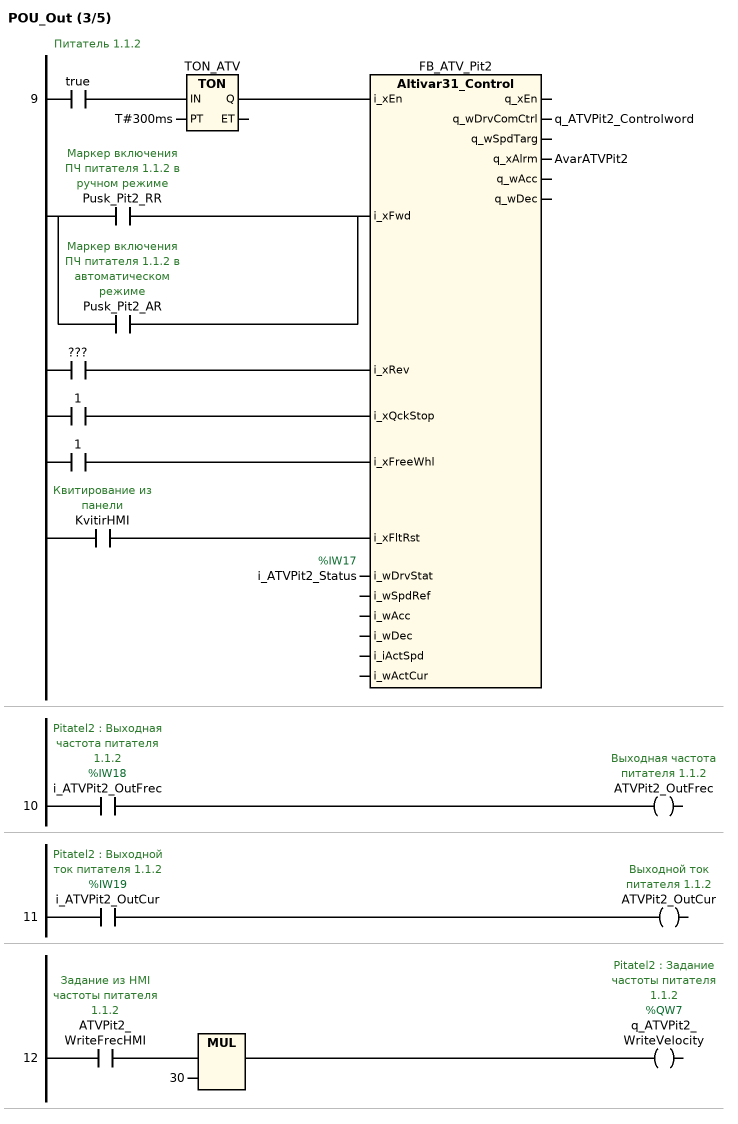
// NETWORK 9
// Питатель 1.1.2
//   Pusk_Pit2_RR: Маркер включения ПЧ питателя 1.1.2 в ручном режиме
//   Pusk_Pit2_AR: Маркер включения ПЧ питателя 1.1.2 в автоматическом режиме
//   KvitirHMI: Квитирование из панели
//   i_ATVPit2_Status: Pitatel2 : | AT %IW17
//   q_ATVPit2_Controlword: Pitatel2 : | AT %QW5
//   AvarATVPit2: Защита ПЧ питателя 1.1.2
TON_ATV(IN := true, PT := T#300ms); // TON
FB_ATV_Pit2(
    i_xEn := TON_ATV.Q,
    i_xFwd := Pusk_Pit2_RR OR Pusk_Pit2_AR,
    i_xQckStop := 1,
    i_xFreeWhl := 1,
    i_xFltRst := KvitirHMI,
    i_wDrvStat := i_ATVPit2_Status,
    q_wDrvComCtrl => q_ATVPit2_Controlword,
    q_xAlrm => AvarATVPit2); // Altivar31_Control

// NETWORK 10
//   i_ATVPit2_OutFrec: Pitatel2 : Выходная частота питателя 1.1.2 | AT %IW18
//   ATVPit2_OutFrec: Выходная частота питателя 1.1.2
ATVPit2_OutFrec := i_ATVPit2_OutFrec;

// NETWORK 11
//   i_ATVPit2_OutCur: Pitatel2 : Выходной ток питателя 1.1.2 | AT %IW19
//   ATVPit2_OutCur: Выходной ток питателя 1.1.2
ATVPit2_OutCur := i_ATVPit2_OutCur;

// NETWORK 12
//   ATVPit2_WriteFrecHMI: Задание из HMI частоты питателя 1.1.2
//   q_ATVPit2_WriteVelocity: Pitatel2 : Задание частоты питателя 1.1.2 | AT %QW7
q_ATVPit2_WriteVelocity := ATVPit2_WriteFrecHMI * 30;

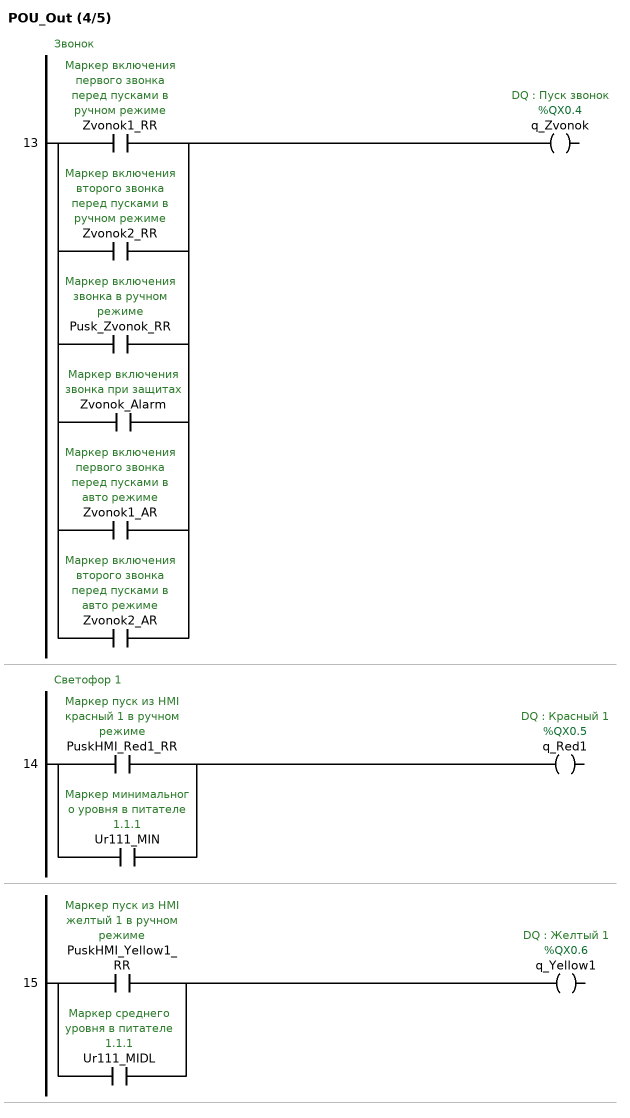
// NETWORK 13
// Звонок
//   Zvonok1_RR: Маркер включения первого звонка перед пусками в ручном режиме
//   Zvonok2_RR: Маркер включения второго звонка перед пусками в ручном режиме
//   Pusk_Zvonok_RR: Маркер включения звонка в ручном режиме
//   Zvonok_Alarm: Маркер включения звонка при защитах
//   Zvonok1_AR: Маркер включения первого звонка перед пусками в авто режиме
//   Zvonok2_AR: Маркер включения второго звонка перед пусками в авто режиме
//   q_Zvonok: DQ : Пуск звонок | AT %QX0.4
q_Zvonok := Zvonok1_RR OR Zvonok2_RR OR Pusk_Zvonok_RR OR Zvonok_Alarm OR Zvonok1_AR OR Zvonok2_AR;

// NETWORK 14
// Светофор 1
//   PuskHMI_Red1_RR: Маркер пуск из HMI красный 1 в ручном режиме
//   Ur111_MIN: Маркер минимального уровня в питателе 1.1.1
//   q_Red1: DQ : Красный 1 | AT %QX0.5
q_Red1 := PuskHMI_Red1_RR OR Ur111_MIN;

// NETWORK 15
//   PuskHMI_Yellow1_RR: Маркер пуск из HMI желтый 1 в ручном режиме
//   Ur111_MIDL: Маркер среднего уровня в питателе 1.1.1
//   q_Yellow1: DQ : Желтый 1 | AT %QX0.6
q_Yellow1 := PuskHMI_Yellow1_RR OR Ur111_MIDL;

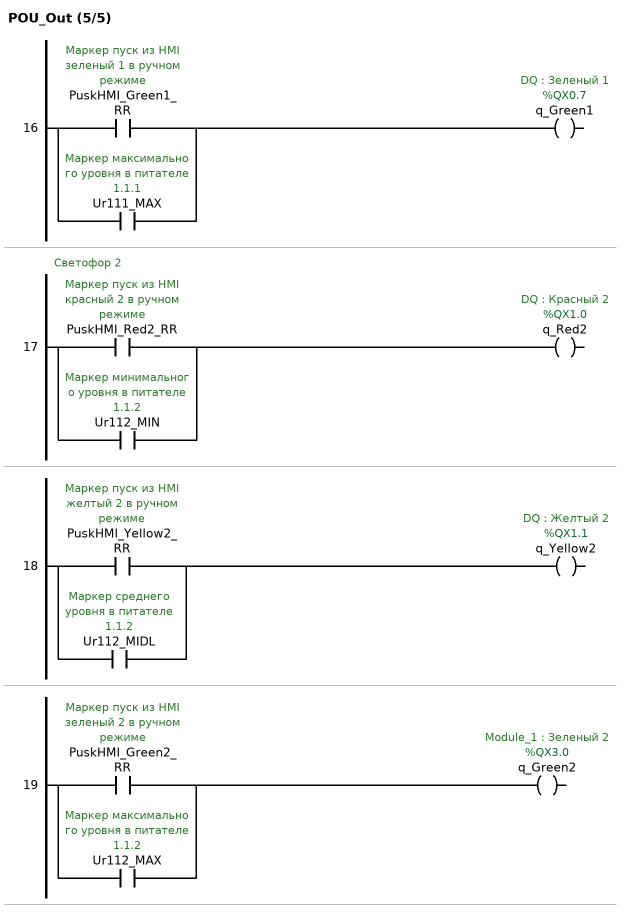
// NETWORK 16
//   PuskHMI_Green1_RR: Маркер пуск из HMI зеленый 1 в ручном режиме
//   Ur111_MAX: Маркер максимального уровня в питателе 1.1.1
//   q_Green1: DQ : Зеленый 1 | AT %QX0.7
q_Green1 := PuskHMI_Green1_RR OR Ur111_MAX;

// NETWORK 17
// Светофор 2
//   PuskHMI_Red2_RR: Маркер пуск из HMI красный 2 в ручном режиме
//   Ur112_MIN: Маркер минимального уровня в питателе 1.1.2
//   q_Red2: DQ : Красный 2 | AT %QX1.0
q_Red2 := PuskHMI_Red2_RR OR Ur112_MIN;

// NETWORK 18
//   PuskHMI_Yellow2_RR: Маркер пуск из HMI желтый 2 в ручном режиме
//   Ur112_MIDL: Маркер среднего уровня в питателе 1.1.2
//   q_Yellow2: DQ : Желтый 2 | AT %QX1.1
q_Yellow2 := PuskHMI_Yellow2_RR OR Ur112_MIDL;

// NETWORK 19
//   PuskHMI_Green2_RR: Маркер пуск из HMI зеленый 2 в ручном режиме
//   Ur112_MAX: Маркер максимального уровня в питателе 1.1.2
//   q_Green2: Module_1 : Зеленый 2 | AT %QX3.0
q_Green2 := PuskHMI_Green2_RR OR Ur112_MAX;

END_PROGRAM

// MyController/Application/POU_Alarm
PROGRAM POU_Alarm
VAR
	RS_Zv: RS;
	// Сброс звонка из HMI
	SbrosZvonka: BOOL;
	SR_AvStop: SR;
	SR_KR2: SR;
	SR_Pit1: SR;
	SR_Pit2: SR;
	SR_K1: SR;
END_VAR
VAR // added by the converter: edge detectors and wires of the graphical bodies
    _ft1 : F_TRIG;
    _rt1, _rt2, _rt3, _rt4 : R_TRIG;
END_VAR

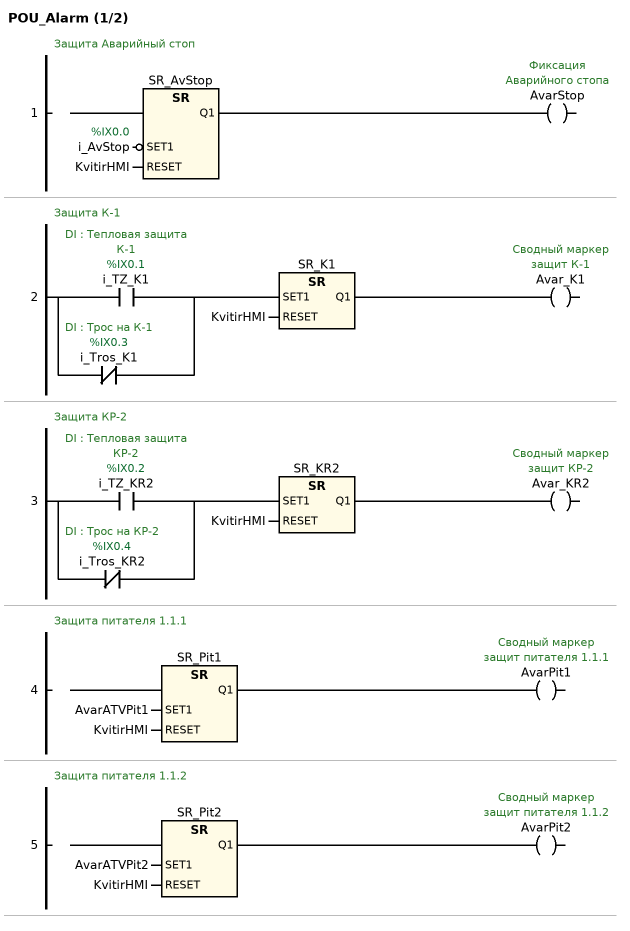
// NETWORK 1
// Защита Аварийный стоп
//   i_AvStop: DI : Аварийный стоп. При отсутствии сигнала | AT %IX0.0
//   KvitirHMI: Квитирование из панели
//   AvarStop: Фиксация Аварийного стопа
SR_AvStop(SET1 := NOT i_AvStop, RESET := KvitirHMI); // SR
AvarStop := SR_AvStop.Q1;

// NETWORK 2
// Защита К-1
//   i_TZ_K1: DI : Тепловая защита К-1 | AT %IX0.1
//   i_Tros_K1: DI : Трос на К-1 | AT %IX0.3
//   KvitirHMI: Квитирование из панели
//   Avar_K1: Сводный маркер защит К-1
SR_K1(SET1 := i_TZ_K1 OR NOT i_Tros_K1, RESET := KvitirHMI); // SR
Avar_K1 := SR_K1.Q1;

// NETWORK 3
// Защита КР-2
//   i_TZ_KR2: DI : Тепловая защита КР-2 | AT %IX0.2
//   i_Tros_KR2: DI : Трос на КР-2 | AT %IX0.4
//   KvitirHMI: Квитирование из панели
//   Avar_KR2: Сводный маркер защит КР-2
SR_KR2(SET1 := i_TZ_KR2 OR NOT i_Tros_KR2, RESET := KvitirHMI); // SR
Avar_KR2 := SR_KR2.Q1;

// NETWORK 4
// Защита питателя 1.1.1
//   AvarATVPit1: Защита ПЧ питателя 1.1.1
//   KvitirHMI: Квитирование из панели
//   AvarPit1: Сводный маркер защит питателя 1.1.1
SR_Pit1(SET1 := AvarATVPit1, RESET := KvitirHMI); // SR
AvarPit1 := SR_Pit1.Q1;

// NETWORK 5
// Защита питателя 1.1.2
//   AvarATVPit2: Защита ПЧ питателя 1.1.2
//   KvitirHMI: Квитирование из панели
//   AvarPit2: Сводный маркер защит питателя 1.1.2
SR_Pit2(SET1 := AvarATVPit2, RESET := KvitirHMI); // SR
AvarPit2 := SR_Pit2.Q1;

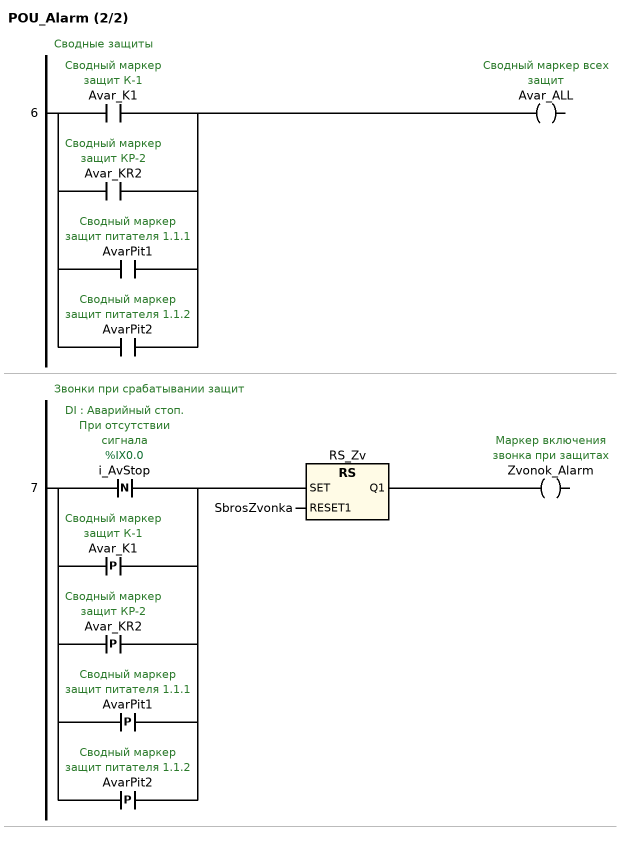
// NETWORK 6
// Сводные защиты
//   Avar_K1: Сводный маркер защит К-1
//   Avar_KR2: Сводный маркер защит КР-2
//   AvarPit1: Сводный маркер защит питателя 1.1.1
//   AvarPit2: Сводный маркер защит питателя 1.1.2
//   Avar_ALL: Сводный маркер всех защит
Avar_ALL := Avar_K1 OR Avar_KR2 OR AvarPit1 OR AvarPit2;

// NETWORK 7
// Звонки при срабатывании защит
//   i_AvStop: DI : Аварийный стоп. При отсутствии сигнала | AT %IX0.0
//   Avar_K1: Сводный маркер защит К-1
//   Avar_KR2: Сводный маркер защит КР-2
//   AvarPit1: Сводный маркер защит питателя 1.1.1
//   AvarPit2: Сводный маркер защит питателя 1.1.2
//   SbrosZvonka: Сброс звонка из HMI
//   Zvonok_Alarm: Маркер включения звонка при защитах
_ft1(CLK := i_AvStop);
_rt1(CLK := Avar_K1);
_rt2(CLK := Avar_KR2);
_rt3(CLK := AvarPit1);
_rt4(CLK := AvarPit2);
RS_Zv(SET := _ft1.Q OR _rt1.Q OR _rt2.Q OR _rt3.Q OR _rt4.Q, RESET1 := SbrosZvonka); // RS
Zvonok_Alarm := RS_Zv.Q1;

END_PROGRAM

// MyController/Application/POU_testing
PROGRAM POU_testing
VAR
	ONBOARD_ON_OFF: BOOL;
	ONBOARD_0_1: BOOL;
	EXTMOD_ON_OFF: BOOL;
	EXTMOD_0_1: BOOL;
END_VAR
VAR // added by the converter: edge detectors and wires of the graphical bodies
    _rt1, _rt2, _rt3, _rt4, _rt5, _rt6 : R_TRIG;
    _w1, _w2 : BOOL;
    _ft1, _ft2, _ft3, _ft4 : F_TRIG;
END_VAR

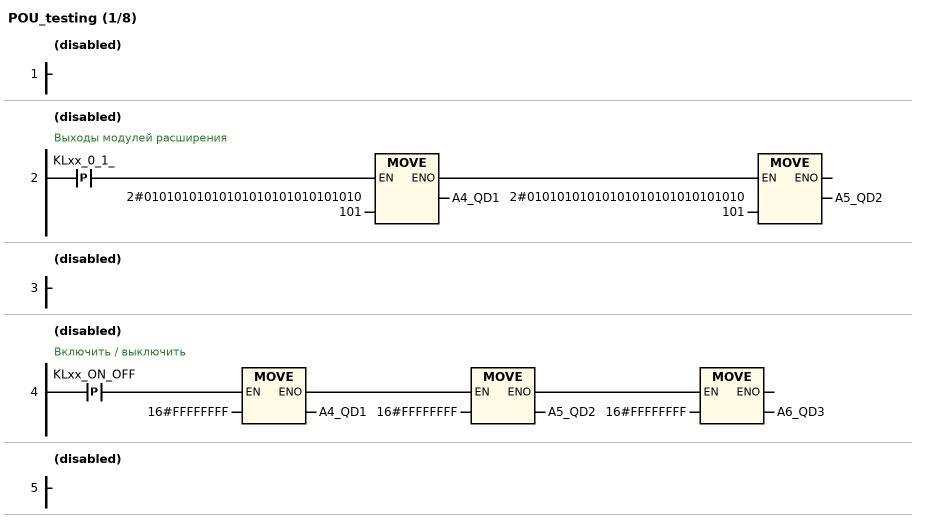
// NETWORK 1 (disabled)

// NETWORK 2 (disabled)
// Выходы модулей расширения
// _rt1(CLK := KLxx_0_1_);
// _w1 := _rt1.Q;
// IF _w1 THEN A4_QD1 := 2#01010101010101010101010101010101; END_IF
// IF _w1 THEN A5_QD2 := 2#01010101010101010101010101010101; END_IF

// NETWORK 3 (disabled)

// NETWORK 4 (disabled)
// Включить / выключить
// _rt2(CLK := KLxx_ON_OFF);
// _w2 := _rt2.Q;
// IF _w2 THEN A4_QD1 := 16#FFFFFFFF; END_IF
// IF _w2 THEN A5_QD2 := 16#FFFFFFFF; END_IF
// IF _w2 THEN A6_QD3 := 16#FFFFFFFF; END_IF

// NETWORK 5 (disabled)

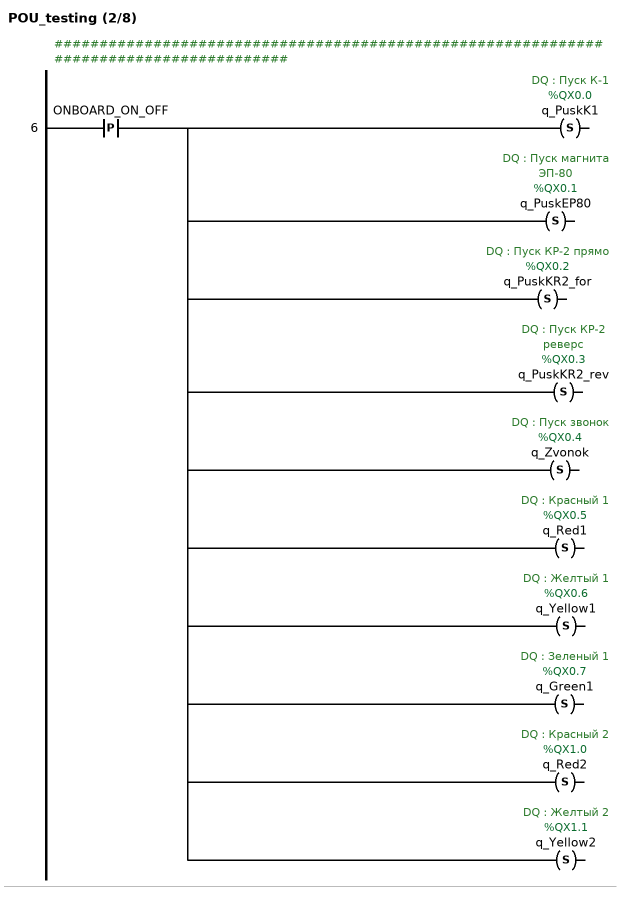
// NETWORK 6
// #######################################################################################
//   q_PuskK1: DQ : Пуск К-1 | AT %QX0.0
//   q_PuskEP80: DQ : Пуск магнита ЭП-80 | AT %QX0.1
//   q_PuskKR2_for: DQ : Пуск КР-2 прямо | AT %QX0.2
//   q_PuskKR2_rev: DQ : Пуск КР-2 реверс | AT %QX0.3
//   q_Zvonok: DQ : Пуск звонок | AT %QX0.4
//   q_Red1: DQ : Красный 1 | AT %QX0.5
//   q_Yellow1: DQ : Желтый 1 | AT %QX0.6
//   q_Green1: DQ : Зеленый 1 | AT %QX0.7
//   q_Red2: DQ : Красный 2 | AT %QX1.0
//   q_Yellow2: DQ : Желтый 2 | AT %QX1.1
_rt3(CLK := ONBOARD_ON_OFF);
q_PuskK1 S= _rt3.Q;
q_PuskEP80 S= _rt3.Q;
q_PuskKR2_for S= _rt3.Q;
q_PuskKR2_rev S= _rt3.Q;
q_Zvonok S= _rt3.Q;
q_Red1 S= _rt3.Q;
q_Yellow1 S= _rt3.Q;
q_Green1 S= _rt3.Q;
q_Red2 S= _rt3.Q;
q_Yellow2 S= _rt3.Q;

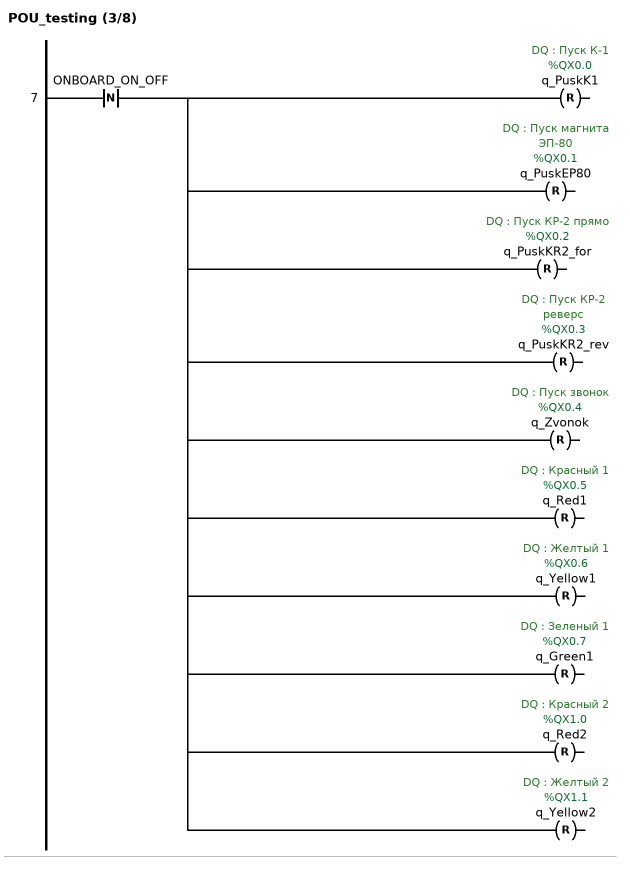
// NETWORK 7
//   q_PuskK1: DQ : Пуск К-1 | AT %QX0.0
//   q_PuskEP80: DQ : Пуск магнита ЭП-80 | AT %QX0.1
//   q_PuskKR2_for: DQ : Пуск КР-2 прямо | AT %QX0.2
//   q_PuskKR2_rev: DQ : Пуск КР-2 реверс | AT %QX0.3
//   q_Zvonok: DQ : Пуск звонок | AT %QX0.4
//   q_Red1: DQ : Красный 1 | AT %QX0.5
//   q_Yellow1: DQ : Желтый 1 | AT %QX0.6
//   q_Green1: DQ : Зеленый 1 | AT %QX0.7
//   q_Red2: DQ : Красный 2 | AT %QX1.0
//   q_Yellow2: DQ : Желтый 2 | AT %QX1.1
_ft1(CLK := ONBOARD_ON_OFF);
q_PuskK1 R= _ft1.Q;
q_PuskEP80 R= _ft1.Q;
q_PuskKR2_for R= _ft1.Q;
q_PuskKR2_rev R= _ft1.Q;
q_Zvonok R= _ft1.Q;
q_Red1 R= _ft1.Q;
q_Yellow1 R= _ft1.Q;
q_Green1 R= _ft1.Q;
q_Red2 R= _ft1.Q;
q_Yellow2 R= _ft1.Q;

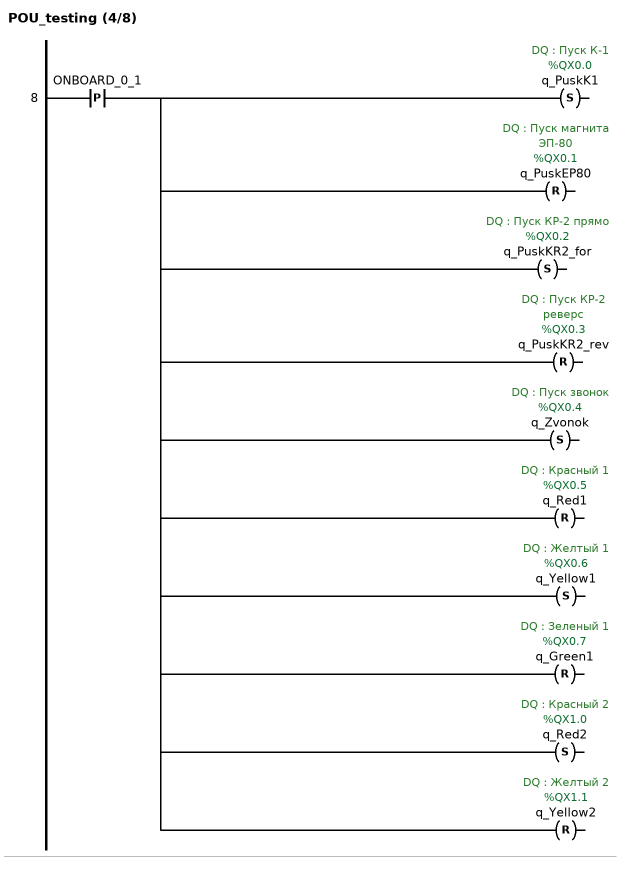
// NETWORK 8
//   q_PuskK1: DQ : Пуск К-1 | AT %QX0.0
//   q_PuskEP80: DQ : Пуск магнита ЭП-80 | AT %QX0.1
//   q_PuskKR2_for: DQ : Пуск КР-2 прямо | AT %QX0.2
//   q_PuskKR2_rev: DQ : Пуск КР-2 реверс | AT %QX0.3
//   q_Zvonok: DQ : Пуск звонок | AT %QX0.4
//   q_Red1: DQ : Красный 1 | AT %QX0.5
//   q_Yellow1: DQ : Желтый 1 | AT %QX0.6
//   q_Green1: DQ : Зеленый 1 | AT %QX0.7
//   q_Red2: DQ : Красный 2 | AT %QX1.0
//   q_Yellow2: DQ : Желтый 2 | AT %QX1.1
_rt4(CLK := ONBOARD_0_1);
q_PuskK1 S= _rt4.Q;
q_PuskEP80 R= _rt4.Q;
q_PuskKR2_for S= _rt4.Q;
q_PuskKR2_rev R= _rt4.Q;
q_Zvonok S= _rt4.Q;
q_Red1 R= _rt4.Q;
q_Yellow1 S= _rt4.Q;
q_Green1 R= _rt4.Q;
q_Red2 S= _rt4.Q;
q_Yellow2 R= _rt4.Q;

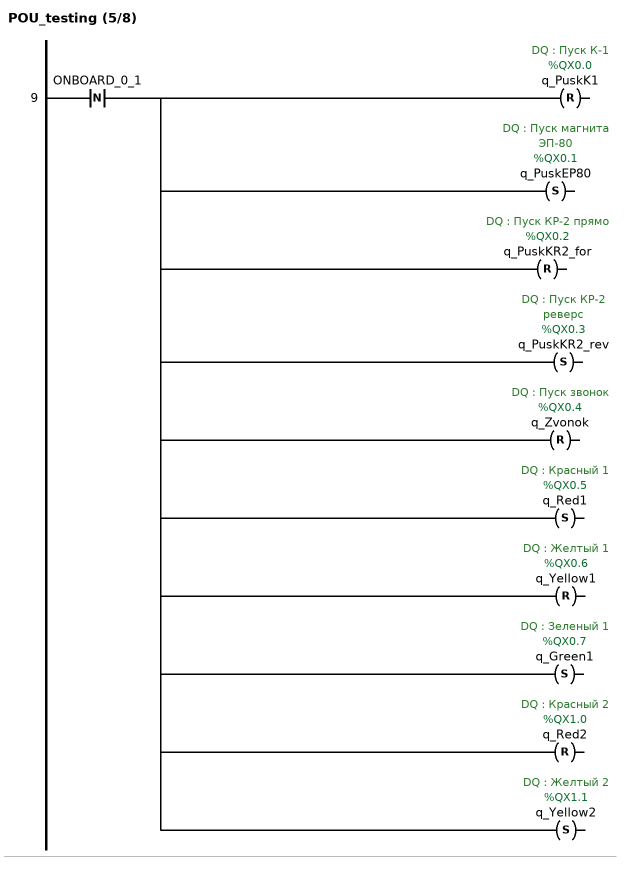
// NETWORK 9
//   q_PuskK1: DQ : Пуск К-1 | AT %QX0.0
//   q_PuskEP80: DQ : Пуск магнита ЭП-80 | AT %QX0.1
//   q_PuskKR2_for: DQ : Пуск КР-2 прямо | AT %QX0.2
//   q_PuskKR2_rev: DQ : Пуск КР-2 реверс | AT %QX0.3
//   q_Zvonok: DQ : Пуск звонок | AT %QX0.4
//   q_Red1: DQ : Красный 1 | AT %QX0.5
//   q_Yellow1: DQ : Желтый 1 | AT %QX0.6
//   q_Green1: DQ : Зеленый 1 | AT %QX0.7
//   q_Red2: DQ : Красный 2 | AT %QX1.0
//   q_Yellow2: DQ : Желтый 2 | AT %QX1.1
_ft2(CLK := ONBOARD_0_1);
q_PuskK1 R= _ft2.Q;
q_PuskEP80 S= _ft2.Q;
q_PuskKR2_for R= _ft2.Q;
q_PuskKR2_rev S= _ft2.Q;
q_Zvonok R= _ft2.Q;
q_Red1 S= _ft2.Q;
q_Yellow1 R= _ft2.Q;
q_Green1 S= _ft2.Q;
q_Red2 R= _ft2.Q;
q_Yellow2 S= _ft2.Q;

